TEST_FINISHED();
END_METHOD

METHOD PRIVATE Test_ANY_STRING_Differ_2
VAR
    a : STRING := 'This is a string';
    b : STRING := 'This is b string';
END_VAR
TEST('Test_ANY_STRING_Differ_2');

AssertEquals(Expected := a,
             Actual := b,
             Message := 'Values differ');

TEST_FINISHED();
END_METHOD

METHOD PRIVATE Test_ANY_STRING_Equals
VAR
    a : STRING := 'Hello there';
    b : STRING := 'Hello there';
END_VAR
TEST('Test_ANY_STRING_Equals');

AssertEquals(Expected := a,
             Actual := b,
             Message := 'Values differ');

TEST_FINISHED();
END_METHOD

METHOD PRIVATE Test_ANY_TIME_Differ
VAR
    a : TIME := T#12H34M15S10MS;
    b : TIME := T#11H34M13S244MS;
END_VAR
TEST('Test_ANY_TIME_Differ');

AssertEquals(Expected := a,
             Actual := b,
             Message := 'Values differ');

TEST_FINISHED();
END_METHOD

METHOD PRIVATE Test_ANY_TIME_Equals
VAR
    a : TIME := T#11H34M13S244MS;
    b : TIME := T#11H34M13S244MS;
END_VAR
TEST('Test_ANY_TIME_Equals');

AssertEquals(Expected := a,
             Actual := b,
             Message := 'Values differ');

TEST_FINISHED();
END_METHOD

METHOD PRIVATE Test_ANY_TIME_OF_DAY_Differ
VAR
    a : TIME_OF_DAY := TIME_OF_DAY#15:36:30.123;
    b : TIME_OF_DAY := TIME_OF_DAY#06:21:11.492;
END_VAR
TEST('Test_ANY_TIME_OF_DAY_Differ');

AssertEquals(Expected := a,
             Actual := b,
             Message := 'Values differ');

TEST_FINISHED();
END_METHOD

METHOD PRIVATE Test_ANY_TIME_OF_DAY_Equals
VAR
    a : TIME_OF_DAY := TIME_OF_DAY#06:21:11.492;
    b : TIME_OF_DAY := TIME_OF_DAY#06:21:11.492;
END_VAR
TEST('Test_ANY_TIME_OF_DAY_Equals');

AssertEquals(Expected := a,
             Actual := b,
             Message := 'Values differ');

TEST_FINISHED();
END_METHOD

METHOD PRIVATE Test_ANY_UDINT_Differ
VAR
    a : UDINT := 34124214;
    b : UDINT := 52343244;
END_VAR
TEST('Test_ANY_UDINT_Differ');

AssertEquals(Expected := a,
             Actual := b,
             Message := 'Values differ');

TEST_FINISHED();
END_METHOD

METHOD PRIVATE Test_ANY_UDINT_Equals
VAR
    a : UDINT := 21845123;
    b : UDINT := 21845123;
END_VAR
TEST('Test_ANY_UDINT_Equals');

AssertEquals(Expected := a,
             Actual := b,
             Message := 'Values differ');

TEST_FINISHED();
END_METHOD

METHOD PRIVATE Test_ANY_UINT_Differ
VAR
    a : UINT := 64322;
    b : UINT := 32312;
END_VAR
TEST('Test_ANY_UINT_Differ');

AssertEquals(Expected := a,
             Actual := b,
             Message := 'Values differ');

TEST_FINISHED();
END_METHOD

METHOD PRIVATE Test_ANY_UINT_Equals
VAR
    a : UINT := 65535;
    b : UINT := 65535;
END_VAR
TEST('Test_ANY_UINT_Equals');

AssertEquals(Expected := a,
             Actual := b,
             Message := 'Values differ');

TEST_FINISHED();
END_METHOD

METHOD PRIVATE Test_ANY_ULINT_Differ
VAR
    a : ULINT := 10000;
    b : ULINT := 53685437234;
END_VAR
TEST('Test_ANY_ULINT_Differ');

AssertEquals(Expected := a,
             Actual := b,
             Message := 'Values differ');

TEST_FINISHED();
END_METHOD

METHOD PRIVATE Test_ANY_ULINT_Equals
VAR
    a : ULINT := 45683838383;
    b : ULINT := 45683838383;
END_VAR
TEST('Test_ANY_ULINT_Equals');

AssertEquals(Expected := a,
             Actual := b,
             Message := 'Values differ');

TEST_FINISHED();
END_METHOD

METHOD PRIVATE Test_ANY_USINT_Differ
VAR
    a : USINT := 3;
    b : USINT := 7;
END_VAR
TEST('Test_ANY_USINT_Differ');

AssertEquals(Expected := a,
             Actual := b,
             Message := 'Values differ');

TEST_FINISHED();
END_METHOD

METHOD PRIVATE Test_ANY_USINT_Equals
VAR
    a : USINT := 5;
    b : USINT := 5;
END_VAR
TEST('Test_ANY_USINT_Equals');

AssertEquals(Expected := a,
             Actual := b,
             Message := 'Values differ');

TEST_FINISHED();
END_METHOD

METHOD PRIVATE Test_ANY_WORD_Differ
VAR
    a : WORD := 16#EF01;
    b : WORD := 16#2345;
END_VAR
TEST('Test_ANY_WORD_Differ');

AssertEquals(Expected := a,
             Actual := b,
             Message := 'Values differ');

TEST_FINISHED();
END_METHOD

METHOD PRIVATE Test_ANY_WORD_Equals
VAR
    a : WORD := 16#ABCD;
    b : WORD := 16#ABCD;
END_VAR
TEST('Test_ANY_WORD_Equals');

AssertEquals(Expected := a,
             Actual := b,
             Message := 'Values differ');

TEST_FINISHED();
END_METHOD

METHOD PRIVATE Test_ANY_WSTRING_Differ
VAR
    a : WSTRING := "äö";
    b : WSTRING := "æå";
END_VAR
TEST('Test_ANY_WSTRING_Differ');

AssertEquals(Expected := a,
             Actual := b,
             Message := 'Values differ');

TEST_FINISHED();
END_METHOD

METHOD PRIVATE Test_ANY_WSTRING_Differ_2
VAR
    a : WSTRING := "äö◦";
    b : WSTRING := "æå";
END_VAR
TEST('Test_ANY_WSTRING_Differ_2');

AssertEquals(Expected := a,
             Actual := b,
             Message := 'Values differ');

TEST_FINISHED();
END_METHOD

METHOD PRIVATE Test_ANY_WSTRING_Equals
VAR
    a : WSTRING := "ĠĦ";
    b : WSTRING := "ĠĦ";
END_VAR
TEST('Test_ANY_WSTRING_Equals');

AssertEquals(Expected := a,
             Actual := b,
             Message := 'Values differ');

TEST_FINISHED();
END_METHOD

END_FUNCTION_BLOCK

// ---- Test/FB_AssertEveryFailedTestTwiceArrayVersion.TcPOU
(*
    In this testsuite we are running the same testcase over two cycles, and thus calling
    every assert method twice. This is in order to verify that we don't print every FAILED assert twice.
    With this version we are doing it with arrays.
*)
FUNCTION_BLOCK FB_AssertEveryFailedTestTwiceArrayVersion EXTENDS TcUnit.FB_TestSuite
VAR
    AssertCount : USINT := 0;
END_VAR

TwiceAssertCall_Arrays();

METHOD PRIVATE TwiceAssertCall_Arrays
VAR
    aBOOL : ARRAY[0..5] OF BOOL := [TRUE, TRUE, FALSE, TRUE, FALSE, TRUE];
    bBOOL : ARRAY[0..5] OF BOOL := [TRUE, TRUE, TRUE, TRUE, FALSE, FALSE];

    aBYTE : ARRAY[0..3] OF BYTE := [16#AB, 16#AA, 16#BB, 16#89];
    bBYTE : ARRAY[0..3] OF BYTE := [16#AB, 16#CD, 16#BB, 16#89];

    aDINT : ARRAY[3..5] OF DINT := [-4746, -2147483645, 0];
    bDINT : ARRAY[3..5] OF DINT := [-4746, -2147483641, 0];

    aDWORD : ARRAY[-2..1] OF DWORD := [16#6789ABCD, 16#EFAA2346, 16#ABABABAB, 16#EEEEEEEE];
    bDWORD : ARRAY[-2..1] OF DWORD := [16#6789ABCD, 16#EF012345, 16#ABABABAB, 16#EEEEEEEE];

    aINT : ARRAY[-8..-6] OF INT := [42, -23, -32768];
    bINT : ARRAY[1..3] OF INT := [42, 24, -32768];

    aLINT : ARRAY[-1..1] OF LINT := [9_223_372_036_854_775_807, -9_223_372_036_853_775_808, 55];
    bLINT : ARRAY[4..6] OF LINT := [9_223_372_036_854_775_807, -9_223_372_036_854_775_808, 55];

    aLREAL : ARRAY[-2..1] OF LREAL := [3.55, 7.88, 2.44];
    bLREAL : ARRAY[-1..2] OF LREAL := [3.56, 7.99, 2.44];

    aLREAL2d : ARRAY[0..1, 0..1] OF LREAL := [4.44, 5.75, 6.96, 7.77];
    bLREAL2d : ARRAY[0..1, 0..1] OF LREAL := [4.45, 5.75, 6.68, 7.77];

    aLREAL3d : ARRAY[0..1, 0..1, 0..1] OF LREAL := [1.0, 2.0, 3.0, 4.0, 5.0, 6.0, 7.0, 8.0];
    bLREAL3d : ARRAY[0..1, 0..1, 0..1] OF LREAL := [1.0, 2.0, 3.0, 4.0, 5.0, 6.4, 7.0, 8.0];

    aLWORD : ARRAY[1..1] OF LWORD := [16#EDCBA09876543210];
    bLWORD : ARRAY[1..1] OF LWORD := [16#01234567890ABCDE];

    aREAL : ARRAY[0..2] OF REAL := [6.55000001, 3.54, 2.44001];
    bREAL : ARRAY[0..2] OF REAL := [6.55, 3.54, 2.44003];

    aREAL2d : ARRAY[0..1, 0..1] OF REAL := [4.45, 5.75, 6.960001, 7.7701];
    bREAL2d : ARRAY[0..1, 0..1] OF REAL := [4.45, 5.75, 6.960002, 7.7703];

    aREAL3d : ARRAY[0..1, 0..1, 0..1] OF REAL := [1.0, 2.0, 3.0, 4.01, 5.0, 6.0, 7.0, 8.0];
    bREAL3d : ARRAY[0..1, 0..1, 0..1] OF REAL := [1.0, 2.0, 3.0, 4.021, 5.0, 6.0, 7.0, 8.0];

    aSINT : ARRAY[0..0] OF SINT := [-128];
    bSINT : ARRAY[0..0] OF SINT := [127];

    aUDINT : ARRAY[-5..-4] OF UDINT := [4294967295, 5];
    bUDINT : ARRAY[0..1] OF UDINT := [4294967295, 4];

    aUINT : ARRAY[0..3] OF UINT := [0, 4, 8, 99];
    bUINT : ARRAY[0..3] OF UINT := [0, 4, 8, 12];

    aULINT : ARRAY[0..1] OF ULINT := [3_213_000_444_000, 9_400_000_000_000];
    bULINT : ARRAY[0..1] OF ULINT := [3_213_000_444_000, 18_446_744_073_709_551_615];

    aUSINT : ARRAY[0..10] OF USINT := [0,1,2,3,6(4),5];
    bUSINT : ARRAY[0..10] OF USINT := [0,1,2,3,6(5),6];

    aWORD : ARRAY[1..7] OF WORD := [16#2323, 16#876A, 16#4CD4, 16#F3DC, 16#BBBB, 16#FFFF, 16#1133];
    bWORD : ARRAY[1..7] OF WORD := [16#2323, 16#876A, 16#4CD4, 16#F3DC, 16#BBBB, 16#FFFF, 16#1122];
END_VAR
TEST('TwiceAssertCall_Arrays');

AssertArrayEquals_BOOL(Expecteds := aBOOL,
                       Actuals := bBOOL,
                       Message := 'Not equal BOOL');

AssertArrayEquals_BYTE(Expecteds := aBYTE,
                       Actuals := bBYTE,
                       Message := 'Not equal BYTE');

AssertArrayEquals_DINT(Expecteds := aDINT,
                       Actuals := bDINT,
                       Message := 'Not equal DINT');

AssertArrayEquals_DWORD(Expecteds := aDWORD,
                        Actuals := bDWORD,
                        Message := 'Not equal DWORD');

AssertArrayEquals_INT(Expecteds := aINT,
                      Actuals := bINT,
                      Message := 'Not equal INT');

AssertArrayEquals_LINT(Expecteds := aLINT,
                       Actuals := bLINT,
                       Message := 'Not equal LINT');

AssertArrayEquals_LREAL(Expecteds := aLREAL,
                        Actuals := bLREAL,
                        Delta := 0.1,
                        Message := 'Not equal LREAL');

AssertArray2dEquals_LREAL(Expecteds := aLREAL2d,
                          Actuals := bLREAL2d,
                          Delta := 0.1,
                          Message := 'Not equal LREAL2D');

AssertArray3dEquals_LREAL(Expecteds := aLREAL3d,
                          Actuals := bLREAL3d,
                          Delta := 0.1,
                          Message := 'Not equal LREAL3D');

AssertArrayEquals_LWORD(Expecteds := aLWORD,
                        Actuals := bLWORD,
                        Message := 'Not equal LWORD');

AssertArrayEquals_SINT(Expecteds := aSINT,
                       Actuals := bSINT,
                       Message := 'Not equal SINT');

AssertArrayEquals_REAL(Expecteds := aREAL,
                       Actuals := bREAL,
                       Delta := 0.00001,
                       Message := 'Not equal REAL');

AssertArray2dEquals_REAL(Expecteds := aREAL2d,
                         Actuals := bREAL2d,
                         Delta := 0.0001,
                         Message := 'Not equal REAL2D');

AssertArray3dEquals_REAL(Expecteds := aREAL3d,
                         Actuals := bREAL3d,
                         Delta := 0.01,
                         Message := 'Not equal REAL3D');

AssertArrayEquals_UDINT(Expecteds := aUDINT,
                        Actuals := bUDINT,
                        Message := 'Not equal UDINT');

AssertArrayEquals_UINT(Expecteds := aUINT,
                       Actuals := bUINT,
                       Message := 'Not equal UINT');

AssertArrayEquals_ULINT(Expecteds := aULINT,
                        Actuals := bULINT,
                        Message := 'Not equal ULINT');

AssertArrayEquals_USINT(Expecteds := aUSINT,
                        Actuals := bUSINT,
                        Message := 'Not equal USINT');

AssertArrayEquals_WORD(Expecteds := aWORD,
                       Actuals := bWORD,
                       Message := 'Not equal WORD');

AssertCount := AssertCount + 1;
IF AssertCount = 2 THEN
    TEST_FINISHED();
END_IF
END_METHOD

END_FUNCTION_BLOCK

// ---- Test/FB_AnyToUnionValue.TcPOU
(*
    Tests the free function F_AnyToUnionValue.
*)
FUNCTION_BLOCK FB_AnyToUnionValue EXTENDS TcUnit.FB_TestSuite
VAR
    aBit : BIT := 1; // Only structures and function blocks can have BIT defined
END_VAR

Test_BOOL();
Test_BIT();
Test_BYTE();
Test_WORD();
Test_DWORD();
Test_LWORD();
Test_SINT();
Test_INT();
Test_DINT();
Test_LINT();
Test_USINT();
Test_UINT();
Test_UDINT();
Test_ULINT();
Test_REAL();
Test_LREAL();
Test_STRING();
Test_STRING_2();
Test_WSTRING();
Test_TIME();
Test_DATE();
Test_DATE_AND_TIME();
Test_TIME_OF_DAY();
Test_LTIME();

METHOD PRIVATE Test_BIT
VAR
    Result : U_ExpectedOrActual;
END_VAR
TEST('Test_BIT');

Result := TcUnit.F_AnyToUnionValue(AnySize := SIZEOF(aBit), AnyTypeClass := IBaseLibrary.TYPE_BIT, AnyValue := ADR(aBit));

AssertEquals(Expected := aBit,
             Actual := result.bitExpectedOrActual,
             Message := 'Values differ');

TEST_FINISHED();
END_METHOD

METHOD PRIVATE Test_BOOL
VAR
    a : BOOL := TRUE;
    Result : U_ExpectedOrActual;
END_VAR
TEST('Test_BOOL');

Result := TcUnit.F_AnyToUnionValue(AnySize := SIZEOF(a), AnyTypeClass := IBaseLibrary.TYPE_BOOL, AnyValue := ADR(a));

AssertEquals(Expected := a,
             Actual := result.boolExpectedOrActual,
             Message := 'Values differ');

TEST_FINISHED();
END_METHOD

METHOD PRIVATE Test_BYTE
VAR
    a : BYTE := 16#8A;
    Result : U_ExpectedOrActual;
END_VAR
TEST('Test_BYTE');

Result := TcUnit.F_AnyToUnionValue(AnySize := SIZEOF(a), AnyTypeClass := IBaseLibrary.TYPE_BYTE, AnyValue := ADR(a));

AssertEquals(Expected := a,
             Actual := result.byteExpectedOrActual,
             Message := 'Values differ');

TEST_FINISHED();
END_METHOD

METHOD PRIVATE Test_DATE
VAR
    a : DATE := D#2106-02-05;
    Result : U_ExpectedOrActual;
END_VAR
TEST('Test_DATE');

Result := TcUnit.F_AnyToUnionValue(AnySize := SIZEOF(a), AnyTypeClass := IBaseLibrary.TYPE_DATE, AnyValue := ADR(a));

AssertEquals(Expected := a,
             Actual := result.dateExpectedOrActual,
             Message := 'Values differ');

TEST_FINISHED();
END_METHOD

METHOD PRIVATE Test_DATE_AND_TIME
VAR
    a : DATE_AND_TIME := DT#2106-02-06-06:28:15;
    Result : U_ExpectedOrActual;
END_VAR
TEST('Test_DATE_AND_TIME');

Result := TcUnit.F_AnyToUnionValue(AnySize := SIZEOF(a), AnyTypeClass := IBaseLibrary.TYPE_DATEANDTIME, AnyValue := ADR(a));

AssertEquals(Expected := a,
             Actual := result.dateandtimeExpectedOrActual,
             Message := 'Values differ');

TEST_FINISHED();
END_METHOD

METHOD PRIVATE Test_DINT
VAR
    a : DINT := 143251;
    Result : U_ExpectedOrActual;
END_VAR
TEST('Test_DINT');

Result := TcUnit.F_AnyToUnionValue(AnySize := SIZEOF(a), AnyTypeClass := IBaseLibrary.TYPE_DINT, AnyValue := ADR(a));

AssertEquals(Expected := a,
             Actual := result.dintExpectedOrActual,
             Message := 'Values differ');

TEST_FINISHED();
END_METHOD

METHOD PRIVATE Test_DWORD
VAR
    a : DWORD := 16#3456CDEF;
    Result : U_ExpectedOrActual;
END_VAR
TEST('Test_DWORD');

Result := TcUnit.F_AnyToUnionValue(AnySize := SIZEOF(a), AnyTypeClass := IBaseLibrary.TYPE_DWORD, AnyValue := ADR(a));

AssertEquals(Expected := a,
             Actual := result.dwordExpectedOrActual,
             Message := 'Values differ');

TEST_FINISHED();
END_METHOD

METHOD PRIVATE Test_INT
VAR
    a : INT := -32000;
    Result : U_ExpectedOrActual;
END_VAR
TEST('Test_INT');

Result := TcUnit.F_AnyToUnionValue(AnySize := SIZEOF(a), AnyTypeClass := IBaseLibrary.TYPE_INT, AnyValue := ADR(a));

AssertEquals(Expected := a,
             Actual := result.intExpectedOrActual,
             Message := 'Values differ');

TEST_FINISHED();
END_METHOD

METHOD PRIVATE Test_LINT
VAR
    a : LINT := -31243145;
    Result : U_ExpectedOrActual;
END_VAR
TEST('Test_LINT');

Result := TcUnit.F_AnyToUnionValue(AnySize := SIZEOF(a), AnyTypeClass := IBaseLibrary.TYPE_LINT, AnyValue := ADR(a));

AssertEquals(Expected := a,
             Actual := result.lintExpectedOrActual,
             Message := 'Values differ');

TEST_FINISHED();
END_METHOD

METHOD PRIVATE Test_LREAL
VAR
    a : LREAL := 43123923124.745423;
    Result : U_ExpectedOrActual;
END_VAR
TEST('Test_LREAL');

Result := TcUnit.F_AnyToUnionValue(AnySize := SIZEOF(a), AnyTypeClass := IBaseLibrary.TYPE_LREAL, AnyValue := ADR(a));

AssertEquals(Expected := a,
             Actual := result.lrealExpectedOrActual,
             Message := 'Values differ');

TEST_FINISHED();
END_METHOD

METHOD PRIVATE Test_LTIME
VAR
    a : LTIME := LTIME#213502D23H34M33S709MS551US615NS;
    Result : U_ExpectedOrActual;
END_VAR
TEST('Test_LTIME');

Result := TcUnit.F_AnyToUnionValue(AnySize := SIZEOF(a), AnyTypeClass := IBaseLibrary.TYPE_LTIME, AnyValue := ADR(a));

AssertEquals(Expected := a,
             Actual := result.ltimeExpectedOrActual,
             Message := 'Values differ');

TEST_FINISHED();
END_METHOD

METHOD PRIVATE Test_LWORD
VAR
    a : LWORD := 16#456CDEF987654321;
    Result : U_ExpectedOrActual;
END_VAR
TEST('Test_LWORD');

Result := TcUnit.F_AnyToUnionValue(AnySize := SIZEOF(a), AnyTypeClass := IBaseLibrary.TYPE_LWORD, AnyValue := ADR(a));

AssertEquals(Expected := a,
             Actual := result.lwordExpectedOrActual,
             Message := 'Values differ');

TEST_FINISHED();
END_METHOD

METHOD PRIVATE Test_REAL
VAR
    a : REAL := 431239.423;
    Result : U_ExpectedOrActual;
END_VAR
TEST('Test_REAL');

Result := TcUnit.F_AnyToUnionValue(AnySize := SIZEOF(a), AnyTypeClass := IBaseLibrary.TYPE_REAL, AnyValue := ADR(a));

AssertEquals(Expected := a,
             Actual := result.realExpectedOrActual,
             Message := 'Values differ');

TEST_FINISHED();
END_METHOD

METHOD PRIVATE Test_SINT
VAR
    a : SINT := 100;
    Result : U_ExpectedOrActual;
END_VAR
TEST('Test_SINT');

Result := TcUnit.F_AnyToUnionValue(AnySize := SIZEOF(a), AnyTypeClass := IBaseLibrary.TYPE_SINT, AnyValue := ADR(a));

AssertEquals(Expected := a,
             Actual := result.sintExpectedOrActual,
             Message := 'Values differ');

TEST_FINISHED();
END_METHOD

METHOD PRIVATE Test_STRING
VAR
    a : STRING := 'This is a random string';
    Result : U_ExpectedOrActual;
END_VAR
TEST('Test_STRING');

Result := TcUnit.F_AnyToUnionValue(AnySize := SIZEOF(a), AnyTypeClass := IBaseLibrary.TYPE_STRING, AnyValue := ADR(a));

AssertEquals(Expected := a,
             Actual := result.stringExpectedOrActual,
             Message := 'Values differ');

TEST_FINISHED();
END_METHOD

METHOD PRIVATE Test_STRING_2
VAR
    a : T_MaxString := '8YNn5KOmPC4dAcpOBdLWnw4WkN126EwXsj65xeurG48gWBepinNaOIKeCVMtWNBSxQWPdtUYiAusDkjMLtQhDtiWbwvmoKcFwiUGDd7pOe0fd52J7hK60oaYAX6VWWmceLJX8utaDVrVzCGXafeZLeHl6jj5enfjg4tfb2WMEBdsBuG2iDKwzwhBLCPqXDnhe5HbemIbtZT7p62OEj2oDqiIYDD6tZdlhBCCelDBx6dbIp32wFm0TpRKsTiwkZ6'; // 255 characters
    Result : U_ExpectedOrActual;
END_VAR
TEST('Test_STRING_2');

Result := TcUnit.F_AnyToUnionValue(AnySize := SIZEOF(a), AnyTypeClass := IBaseLibrary.TYPE_STRING, AnyValue := ADR(a));

AssertEquals(Expected := a,
             Actual := result.stringExpectedOrActual,
             Message := 'Values differ');

TEST_FINISHED();
END_METHOD

METHOD PRIVATE Test_TIME
VAR
    a : TIME := T#15M20S;
    Result : U_ExpectedOrActual;
END_VAR
TEST('Test_TIME');

Result := TcUnit.F_AnyToUnionValue(AnySize := SIZEOF(a), AnyTypeClass := IBaseLibrary.TYPE_TIME, AnyValue := ADR(a));

AssertEquals(Expected := a,
             Actual := result.timeExpectedOrActual,
             Message := 'Values differ');

TEST_FINISHED();
END_METHOD

METHOD PRIVATE Test_TIME_OF_DAY
VAR
    a : TIME_OF_DAY := TOD#15:36:30.123;
    Result : U_ExpectedOrActual;
END_VAR
TEST('Test_TIME_OF_DAY');

Result := TcUnit.F_AnyToUnionValue(AnySize := SIZEOF(a), AnyTypeClass := IBaseLibrary.TYPE_TIMEOFDAY, AnyValue := ADR(a));

AssertEquals(Expected := a,
             Actual := result.timeofdayExpectedOrActual,
             Message := 'Values differ');

TEST_FINISHED();
END_METHOD

METHOD PRIVATE Test_UDINT
VAR
    a : UDINT := 2555;
    Result : U_ExpectedOrActual;
END_VAR
TEST('Test_UDINT');

Result := TcUnit.F_AnyToUnionValue(AnySize := SIZEOF(a), AnyTypeClass := IBaseLibrary.TYPE_UDINT, AnyValue := ADR(a));

AssertEquals(Expected := a,
             Actual := result.udintExpectedOrActual,
             Message := 'Values differ');

TEST_FINISHED();
END_METHOD

METHOD PRIVATE Test_UINT
VAR
    a : UINT := 34523;
    Result : U_ExpectedOrActual;
END_VAR
TEST('Test_UINT');

Result := TcUnit.F_AnyToUnionValue(AnySize := SIZEOF(a), AnyTypeClass := IBaseLibrary.TYPE_UINT, AnyValue := ADR(a));

AssertEquals(Expected := a,
             Actual := result.uintExpectedOrActual,
             Message := 'Values differ');

TEST_FINISHED();
END_METHOD

METHOD PRIVATE Test_ULINT
VAR
    a : ULINT := 25555423;
    Result : U_ExpectedOrActual;
END_VAR
TEST('TEST_ULINT');

Result := TcUnit.F_AnyToUnionValue(AnySize := SIZEOF(a), AnyTypeClass := IBaseLibrary.TYPE_ULINT, AnyValue := ADR(a));

AssertEquals(Expected := a,
             Actual := result.ulintExpectedOrActual,
             Message := 'Values differ');

TEST_FINISHED();
END_METHOD

METHOD PRIVATE Test_USINT
VAR
    a : USINT := 255;
    Result : U_ExpectedOrActual;
END_VAR
TEST('Test_USINT');

Result := TcUnit.F_AnyToUnionValue(AnySize := SIZEOF(a), AnyTypeClass := IBaseLibrary.TYPE_USINT, AnyValue := ADR(a));

AssertEquals(Expected := a,
             Actual := result.usintExpectedOrActual,
             Message := 'Values differ');

TEST_FINISHED();
END_METHOD

METHOD PRIVATE Test_WORD
VAR
    a : WORD := 16#ABCD;
    Result : U_ExpectedOrActual;
END_VAR
TEST('Test_WORD');

Result := TcUnit.F_AnyToUnionValue(AnySize := SIZEOF(a), AnyTypeClass := IBaseLibrary.TYPE_WORD, AnyValue := ADR(a));

AssertEquals(Expected := a,
             Actual := result.wordExpectedOrActual,
             Message := 'Values differ');

TEST_FINISHED();
END_METHOD

METHOD PRIVATE Test_WSTRING
VAR
    a : WSTRING := "åäöĦ";
    Result : U_ExpectedOrActual;
END_VAR
TEST('Test_WSTRING');

Result := TcUnit.F_AnyToUnionValue(AnySize := SIZEOF(a), AnyTypeClass := IBaseLibrary.TYPE_WSTRING, AnyValue := ADR(a));

AssertEquals(Expected := a,
             Actual := result.wstringExpectedOrActual,
             Message := 'Values differ');

TEST_FINISHED();
END_METHOD

END_FUNCTION_BLOCK

// ---- Test/FB_MultipleAssertWithSameParametersInSameCycleWithSameTest.TcPOU
(*
    This test-suite runs several asserts with the same parameters (same expected, actual, message) in the same cycle
    and in the same test.
    The reason we want the framework to support this is that theoretically the user could want to do an assert with the
    same message, in the same test, with the same data values for both expected and actual, although the data that the
    user does the assert on might be from different data sets.
*)
FUNCTION_BLOCK FB_MultipleAssertWithSameParametersInSameCycleWithSameTest EXTENDS TcUnit.FB_TestSuite

Assert_SeveralTimes();

METHOD PRIVATE Assert_SeveralTimes
VAR
    a : DWORD := 16#12345678;
    b : DWORD := 16#90ABCDEF;

    c : DWORD := 16#12345678;
    d : DWORD := 16#90ABCDEF;

    e : DWORD := 16#12345678;
    f : DWORD := 16#90ABCDEF;
END_VAR
TEST('Assert_SeveralTimes');

AssertEquals_DWORD(Expected := a,
                   Actual := b,
                   Message := 'Values differ');

AssertEquals_DWORD(Expected := c,
                   Actual := d,
                   Message := 'Values differ');

AssertEquals_DWORD(Expected := e,
                   Actual := f,
                   Message := 'Values differ');

TEST_FINISHED();
END_METHOD

END_FUNCTION_BLOCK

// ---- Test/FB_MultipleAssertWithSameParametersInDifferentCyclesButWithDifferentTests.TcPOU
(*
    This test-suite runs several asserts with the same parameters (same expected, actual, message), calling the asserts
    in different cycles and using different tests.
    On top of this, we will call new asserts (though with same parameters) in later cycles.
    The reason we want the framework to support this is that theoretically the user could want to do an assert with the
    same message, in different tests, with the same data values for both expected and actual, although the data that the
    user does the assert on might be from different data sets.
*)
FUNCTION_BLOCK FB_MultipleAssertWithSameParametersInDifferentCyclesButWithDifferentTests EXTENDS TcUnit.FB_TestSuite
VAR
    TimerAgain : TON := (PT := T#1S); // Timer to call "AssertSeveralTimesAgain"
    TimerAgainAgain : TON := (PT := T#5S); // Timer to call "AssertSeveralTimesAgainAgain"
    CalledAll : BOOL; // Indication of whether we've called all tests
END_VAR

TimerAgain(IN := TRUE);

Assert_SeveralTimes();

IF TimerAgain.Q THEN
    TimerAgainAgain(IN := TRUE);
    Assert_SeveralTimesAgain();
END_IF

IF TimerAgainAgain.Q THEN
    Assert_SeveralTimesAgainAgain();
    CalledAll := TRUE;
END_IF

METHOD PRIVATE Assert_SeveralTimes
VAR
    a : DWORD := 16#12345678;
    b : DWORD := 16#90ABCDEF;

    c : DWORD := 16#12345678;
    d : DWORD := 16#90ABCDEF;

    e : DWORD := 16#12345678;
    f : DWORD := 16#90ABCDEF;
END_VAR
TEST('Assert_SeveralTimes');

AssertEquals_DWORD(Expected := a,
                   Actual := b,
                   Message := 'Values differ');

AssertEquals_DWORD(Expected := c,
                   Actual := d,
                   Message := 'Values differ');

AssertEquals_DWORD(Expected := e,
                   Actual := f,
                   Message := 'Values differ');

IF CalledAll THEN
    TEST_FINISHED();
END_IF
END_METHOD

METHOD PRIVATE Assert_SeveralTimesAgain
VAR
    a : DWORD := 16#12345678;
    b : DWORD := 16#90ABCDEF;

    c : DWORD := 16#12345678;
    d : DWORD := 16#90ABCDEF;

    e : DWORD := 16#12345678;
    f : DWORD := 16#90ABCDEF;
END_VAR
TEST('Assert_SeveralTimesAgain');

AssertEquals_DWORD(Expected := a,
                   Actual := b,
                   Message := 'Values differ');

AssertEquals_DWORD(Expected := c,
                   Actual := d,
                   Message := 'Values differ');

AssertEquals_DWORD(Expected := e,
                   Actual := f,
                   Message := 'Values differ');

IF CalledAll THEN
    TEST_FINISHED();
END_IF
END_METHOD

METHOD PRIVATE Assert_SeveralTimesAgainAgain
VAR
    a : DWORD := 16#12345678;
    b : DWORD := 16#90ABCDEF;

    c : DWORD := 16#12345678;
    d : DWORD := 16#90ABCDEF;

    e : DWORD := 16#12345678;
    f : DWORD := 16#90ABCDEF;
END_VAR
TEST('Assert_SeveralTimesAgainAgain');

AssertEquals_DWORD(Expected := a,
                   Actual := b,
                   Message := 'Values differ');

AssertEquals_DWORD(Expected := c,
                   Actual := d,
                   Message := 'Values differ');

AssertEquals_DWORD(Expected := e,
                   Actual := f,
                   Message := 'Values differ');

IF CalledAll THEN
    TEST_FINISHED();
END_IF
END_METHOD

END_FUNCTION_BLOCK

// ---- Test/FB_MultipleAssertWithSameParametersInDifferentCyclesAndInSameTest.TcPOU
(*
    This test-suite runs several asserts with the same parameters (same expected, actual, message), calling the asserts
    in different cycles and using the same test.
    On top of this, we will call new asserts (though with same parameters) in later cycles.
    The reason we want the framework to support this is that theoretically the user could want to do an assert with the
    same message, using the same test with the same data values for both expected and actual, and splitting the asserts
    on different cycles.
*)
FUNCTION_BLOCK FB_MultipleAssertWithSameParametersInDifferentCyclesAndInSameTest EXTENDS TcUnit.FB_TestSuite
VAR
    TimerAgain : TON := (PT := T#1S); // Timer to call "AssertSeveralTimesAgain"
    TimerAgainAgain : TON := (PT := T#5S); // Timer to call "AssertSeveralTimesAgainAgain"
    CalledAll : BOOL; // Indication of whether we've called all tests
END_VAR

Assert_SeveralTimes();

METHOD PRIVATE Assert_SeveralTimes
VAR
    a : DWORD := 16#12345678;
    b : DWORD := 16#90ABCDEF;

    c : DWORD := 16#12345678;
    d : DWORD := 16#90ABCDEF;

    e : DWORD := 16#12345678;
    f : DWORD := 16#90ABCDEF;

    g : DWORD := 16#12345678;
    h : DWORD := 16#90ABCDEF;

    i : DWORD := 16#12345678;
    j : DWORD := 16#90ABCDEF;

    k : DWORD := 16#12345678;
    l : DWORD := 16#90ABCDEF;

    m : DWORD := 16#12345678;
    n : DWORD := 16#90ABCDEF;

    o : DWORD := 16#12345678;
    p : DWORD := 16#90ABCDEF;

    q : DWORD := 16#12345678;
    rr : DWORD := 16#90ABCDEF;
END_VAR
TEST('Assert_SeveralTimes');

AssertEquals_DWORD(Expected := a,
                   Actual := b,
                   Message := 'Values differ');
AssertEquals_DWORD(Expected := c,
                   Actual := d,
                   Message := 'Values differ');
AssertEquals_DWORD(Expected := e,
                   Actual := f,
                   Message := 'Values differ');

TimerAgain(IN := TRUE);
IF TimerAgain.Q THEN
    TimerAgainAgain(IN := TRUE);
    AssertEquals_DWORD(Expected := g,
                       Actual := h,
                       Message := 'Values differ');
    AssertEquals_DWORD(Expected := i,
                       Actual := j,
                       Message := 'Values differ');
    AssertEquals_DWORD(Expected := k,
                       Actual := l,
                       Message := 'Values differ');
END_IF

IF TimerAgainAgain.Q THEN
    AssertEquals_DWORD(Expected := m,
                       Actual := n,
                       Message := 'Values differ');
    AssertEquals_DWORD(Expected := o,
                       Actual := p,
                       Message := 'Values differ');
    AssertEquals_DWORD(Expected := q,
                       Actual := rr,
                       Message := 'Values differ');
    CalledAll := TRUE;
    TEST_FINISHED();
END_IF
END_METHOD

END_FUNCTION_BLOCK

// ---- Test/FB_SkipAssertionsWhenFinished.TcPOU
(*
    Contains tests that require multiple cycles:
    - A short test that finishes quickly
        - The assert statements all pass while the test is not finished
        - After the test is finished, the variables change so that the assert statements now fail,
            which shouldn't matter because the test is finished
    - A long test that finishes slowly
        - This test exists so that the entire test suite keeps running after the short test finishes
*)
FUNCTION_BLOCK FB_SkipAssertionsWhenFinished EXTENDS TcUnit.FB_TestSuite
VAR
    ShortTimer : TON := (PT := T#200MS);
    LongTimer : TON := (PT := T#1S);
END_VAR

Test_LongTest(ADR(LongTimer));
Test_ShortTest(ADR(ShortTimer));
Test_AssertImmediatelyAfterFinished();

(*
    Assertions called immediately after (and within the same cycle as) TEST_FINISHED should be
    ignored.
*)
METHOD Test_AssertImmediatelyAfterFinished
TEST('Test_AssertImmediatelyAfterFinished');
TEST_FINISHED();

AssertTrue(FALSE, 'This failing assertion should be skipped because the test is finished');
END_METHOD

METHOD Test_LongTest
VAR_INPUT
    Timer : POINTER TO TON;
END_VAR
TEST('Test_LongTest');

Timer^(IN := TRUE);
IF Timer^.Q THEN
    TEST_FINISHED();
END_IF
END_METHOD

METHOD Test_ShortTest
VAR_INPUT
    Timer : POINTER TO TON;
END_VAR
TEST('Test_ShortTest');

AssertFalse(Timer^.Q, 'This assertion will start to fail after the test is over, but it will be skipped at that point');

Timer^(IN := TRUE);
IF Timer^.Q THEN
    TEST_FINISHED();
END_IF
END_METHOD

END_FUNCTION_BLOCK

// ---- Test/FB_AdjustAssertFailureMessageToMaxAllowedLengthTest.TcPOU
(* This testsuite tests the function block FB_AdjustAssertFailureMessageToMaxAllowedLength
   The total printed message can not be more than 250 characters long.
*)
FUNCTION_BLOCK FB_AdjustAssertFailureMessageToMaxAllowedLengthTest EXTENDS TcUnit.FB_TestSuite

TestInstancePath221CharsExpectShortenedTestInstancePath();
TestInstancePath252CharsExpectTooLongTestInstancePath();
TestInstancePath253CharsExpectTooLongTestInstancePath();
TestInstancePath255CharsExpectTooLongTestInstancePath();

METHOD TestInstancePath221CharsExpectShortenedTestInstancePath
VAR
    AdjustAssertFailureMessageToMaxAllowedLength : FB_AdjustAssertFailureMessageToMaxAllowedLength;

    // @Text-Fixture
    TestInstancePathNameWith221Chars : T_MaxString := 'PRG_TEST.LongInstanceNameLongInstanceNameLongInstanceNameLongInstanceNameLongInstanceNameLongInstanceNameLongInstanceNameLongInstanceNameLongInstanceNameLongInstanceName@LONGTESTNAMELONGTESTNAMELONGTESTNAMELONGTESTNAMELON';
    TooLongTestMessage60Chars : T_MaxString := 'Very long message that is 60 characters long which means tha';

    // @Test-Result-Expected
    // 220 + 32 = 252 (in other words, expected test message should be 32 characters long including '...TestMsg too long'
    TestMessageResultExpected : T_MaxString := 'Very long me...TestMsg too long'; 

    // @Test-Result
    TestInstancePathResult : T_MaxString;
    TestMessageResult : T_MaxString;
END_VAR
TEST('TestInstancePath221CharsExpectShortenedTestInstancePath');

AdjustAssertFailureMessageToMaxAllowedLength(TestInstancePath := TestInstancePathNameWith221Chars,
                                             TestMessage := TooLongTestMessage60Chars,
                                             TestInstancePathProcessed => TestInstancePathResult,
                                             TestMessageProcessed => TestMessageResult);

AssertEquals_STRING(Expected := TestInstancePathNameWith221Chars, // Same test instance path should be expected as the one going in
                    Actual := TestInstancePathResult,
                    'Test instance path not correct');

AssertEquals_STRING(Expected := TestMessageResultExpected,
                    Actual := TestMessageResult,
                    'Test message not correct');

TEST_FINISHED();
END_METHOD

METHOD PRIVATE TestInstancePath252CharsExpectTooLongTestInstancePath
VAR
    AdjustAssertFailureMessageToMaxAllowedLength : FB_AdjustAssertFailureMessageToMaxAllowedLength;

    // @Text-Fixture
    TestInstancePathNameWith252Chars : T_MaxString := 'PRG_TEST.LongInstanceNameLongInstanceNameLongInstanceNameLongInstanceNameLongInstanceNameLongInstanceNameLongInstanceNameLongInstanceNameLongInstanceNameLongInstanceName@LONGTESTNAMELONGTESTNAMELONGTESTNAMELONGTESTNAMELONGTESTNAMELONGTESTNAMELONGTESTNA';
    ShortTestMessage : T_MaxString := 'Very short message';

    // @Test-Result-Expected
    TestInstancePathNameWith252CharsExpectedResult : T_MaxString := 'PRG_TEST.LongInstanceNameLongInstanceNameLongInstanceNameLongInstanceNameLongInstanceNameLongInstanceNameLongInstanceNameLongInstanceNameLongInstanceNameLongInstanceName@LONGTESTNAMELONGTESTNAMELONGTESTNAMELONGTESTNAMELONGTESTNAMELO...TestName too long';
    ShortTestMessageExpectedResult : T_MaxString := '';

    // @Test-Result
    TestInstancePathNameWith252CharsResult : T_MaxString;
    ShortTestMessageResult : T_MaxString;
END_VAR
TEST('TestInstancePath252CharsExpectTooLongTestInstancePath');

AdjustAssertFailureMessageToMaxAllowedLength(TestInstancePath := TestInstancePathNameWith252Chars,
                                             TestMessage := ShortTestMessage,
                                             TestInstancePathProcessed => TestInstancePathNameWith252CharsResult,
                                             TestMessageProcessed => ShortTestMessageResult);

AssertEquals_STRING(Expected := TestInstancePathNameWith252CharsExpectedResult,
                    Actual := TestInstancePathNameWith252CharsResult,
                    'Test instance path not correct');

AssertEquals_STRING(Expected := ShortTestMessageExpectedResult,
                    Actual := ShortTestMessageResult,
                    'Test message not correct');

TEST_FINISHED();
END_METHOD

METHOD PRIVATE TestInstancePath253CharsExpectTooLongTestInstancePath
VAR
    AdjustAssertFailureMessageToMaxAllowedLength : FB_AdjustAssertFailureMessageToMaxAllowedLength;

    // @Text-Fixture
    TestInstancePathNameWith253Chars : T_MaxString := 'PRG_TEST.LongInstanceNameLongInstanceNameLongInstanceNameLongInstanceNameLongInstanceNameLongInstanceNameLongInstanceNameLongInstanceNameLongInstanceNameLongInstanceName@LONGTESTNAMELONGTESTNAMELONGTESTNAMELONGTESTNAMELONGTESTNAMELONGTESTNAMELONGTESTNAM';
    ShortTestMessage : T_MaxString := 'Very short message';

    // @Test-Result-Expected
    TestInstancePathNameWith252CharsExpectedResult : T_MaxString := 'PRG_TEST.LongInstanceNameLongInstanceNameLongInstanceNameLongInstanceNameLongInstanceNameLongInstanceNameLongInstanceNameLongInstanceNameLongInstanceNameLongInstanceName@LONGTESTNAMELONGTESTNAMELONGTESTNAMELONGTESTNAMELONGTESTNAMELO...TestName too long';
    ShortTestMessageExpectedResult : T_MaxString := '';

    // @Test-Result
    TestInstancePathNameWith252CharsResult : T_MaxString;
    ShortTestMessageResult : T_MaxString;
END_VAR
TEST('TestInstancePath253CharsExpectTooLongTestInstancePath');

AdjustAssertFailureMessageToMaxAllowedLength(TestInstancePath := TestInstancePathNameWith253Chars,
                                             TestMessage := ShortTestMessage,
                                             TestInstancePathProcessed => TestInstancePathNameWith252CharsResult,
                                             TestMessageProcessed => ShortTestMessageResult);

AssertEquals_STRING(Expected := TestInstancePathNameWith252CharsExpectedResult,
                    Actual := TestInstancePathNameWith252CharsResult,
                    'Test instance path not correct');

AssertEquals_STRING(Expected := ShortTestMessageExpectedResult,
                    Actual := ShortTestMessageResult,
                    'Test message not correct');

TEST_FINISHED();
END_METHOD

METHOD PRIVATE TestInstancePath255CharsExpectTooLongTestInstancePath
VAR
    AdjustAssertFailureMessageToMaxAllowedLength : FB_AdjustAssertFailureMessageToMaxAllowedLength;

    // @Text-Fixture
    TestInstancePathNameWith255Chars : T_MaxString := 'PRG_TEST.LongInstanceNameLongInstanceNameLongInstanceNameLongInstanceNameLongInstanceNameLongInstanceNameLongInstanceNameLongInstanceNameLongInstanceNameLongInstanceName@LONGTESTNAMELONGTESTNAMELONGTESTNAMELONGTESTNAMELONGTESTNAMELONGTESTNAMELONGTESTNAGAV';
    ShortTestMessage : T_MaxString := 'Very short message';

    // @Test-Result-Expected
    TestInstancePathNameWith252CharsExpectedResult : T_MaxString := 'PRG_TEST.LongInstanceNameLongInstanceNameLongInstanceNameLongInstanceNameLongInstanceNameLongInstanceNameLongInstanceNameLongInstanceNameLongInstanceNameLongInstanceName@LONGTESTNAMELONGTESTNAMELONGTESTNAMELONGTESTNAMELONGTESTNAMELO...TestName too long';
    ShortTestMessageExpectedResult : T_MaxString := '';

    // @Test-Result
    TestInstancePathNameWith252CharsResult : T_MaxString;
    ShortTestMessageResult : T_MaxString;
END_VAR
TEST('TestInstancePath255CharsExpectTooLongTestInstancePath');

AdjustAssertFailureMessageToMaxAllowedLength(TestInstancePath := TestInstancePathNameWith255Chars,
                                             TestMessage := ShortTestMessage,
                                             TestInstancePathProcessed => TestInstancePathNameWith252CharsResult,
                                             TestMessageProcessed => ShortTestMessageResult);

AssertEquals_STRING(Expected := TestInstancePathNameWith252CharsExpectedResult,
                    Actual := TestInstancePathNameWith252CharsResult,
                    'Test instance path not correct');

AssertEquals_STRING(Expected := ShortTestMessageExpectedResult,
                    Actual := ShortTestMessageResult,
                    'Test message not correct');

TEST_FINISHED();
END_METHOD

END_FUNCTION_BLOCK

// ---- Test/FB_EmptyTestSuite.TcPOU
(* This is an empty testsuite with no test cases, so that we can verify that the system still prints the
   test results. *)
FUNCTION_BLOCK FB_EmptyTestSuite EXTENDS TcUnit.FB_TestSuite
VAR
END_VAR

END_FUNCTION_BLOCK

// ---- Test/FB_CheckIfSpecificTestIsFinished.TcPOU
// Verifies that the function IS_TEST_FINISHED('Name') works as intended.
FUNCTION_BLOCK FB_CheckIfSpecificTestIsFinished EXTENDS TcUnit.FB_TestSuite

CheckBeforeAndAfterFinishing();

METHOD CheckBeforeAndAfterFinishing
TEST('CheckBeforeAndAfterFinishing');

AssertEquals_BOOL(Expected := FALSE,
                  Actual := IS_TEST_FINISHED('CheckBeforeAndAfterFinishing'),
                  Message:='Values differ before finishing');

TEST_FINISHED();

AssertEquals_BOOL(Expected := TRUE,
                  Actual := IS_TEST_FINISHED('CheckBeforeAndAfterFinishing'),
                  Message:='Values differ after finishing');
END_METHOD

END_FUNCTION_BLOCK

// ---- Test/FB_WriteProtectedFunctions.TcPOU
// This testsuite tests the WRITE_PROTECTED_* helper functions.
FUNCTION_BLOCK FB_WriteProtectedFunctions EXTENDS TcUnit.FB_TestSuite

Test_WRITE_PROTECTED_BOOL();
Test_WRITE_PROTECTED_BYTE();
Test_WRITE_PROTECTED_DATE();
Test_WRITE_PROTECTED_DATE_AND_TIME();
Test_WRITE_PROTECTED_DINT();
Test_WRITE_PROTECTED_DWORD();
Test_WRITE_PROTECTED_INT();
TEST_WRITE_PROTECTED_LINT();
Test_WRITE_PROTECTED_LREAL();
Test_WRITE_PROTECTED_LWORD();
Test_WRITE_PROTECTED_REAL();
Test_WRITE_PROTECTED_SINT();
Test_WRITE_PROTECTED_STRING();
Test_WRITE_PROTECTED_TIME();
Test_WRITE_PROTECTED_TIME_OF_DAY();
Test_WRITE_PROTECTED_UDINT();
Test_WRITE_PROTECTED_UINT();
Test_WRITE_PROTECTED_USINT();
Test_WRITE_PROTECTED_ULINT();
Test_WRITE_PROTECTED_WORD();
Test_WRITE_PROTECTED_WSTRING();

METHOD Test_WRITE_PROTECTED_BOOL
VAR
    ProtectedVariables : FB_ProtectedVariables;
END_VAR
TEST('Test_WRITE_PROTECTED_BOOL');

WRITE_PROTECTED_BOOL(ADR(ProtectedVariables.InputBOOL), TRUE);
AssertEquals_BOOL(TRUE, ProtectedVariables.InputBOOL, 'Overwriting protected InputBOOL');

WRITE_PROTECTED_BOOL(ADR(ProtectedVariables.VarBOOL), TRUE);
AssertEquals_BOOL(TRUE, ProtectedVariables.VarBOOL, 'Overwriting protected VarBOOL');

TEST_FINISHED();
END_METHOD

METHOD Test_WRITE_PROTECTED_BYTE
VAR
    ProtectedVariables : FB_ProtectedVariables;
END_VAR
TEST('Test_WRITE_PROTECTED_BYTE');

WRITE_PROTECTED_BYTE(ADR(ProtectedVariables.InputBYTE), 1);
AssertEquals_BYTE(1, ProtectedVariables.InputBYTE, 'Overwriting protected InputBYTE');

WRITE_PROTECTED_BYTE(ADR(ProtectedVariables.VarBYTE), 1);
AssertEquals_BYTE(1, ProtectedVariables.VarBYTE, 'Overwriting protected VarBYTE');

TEST_FINISHED();
END_METHOD

METHOD Test_WRITE_PROTECTED_DATE
VAR
    ProtectedVariables : FB_ProtectedVariables;
END_VAR
TEST('Test_WRITE_PROTECTED_DATE');

WRITE_PROTECTED_DATE(ADR(ProtectedVariables.InputDATE), D#2000-01-01);
AssertEquals_DATE(D#2000-01-01, ProtectedVariables.InputDATE, 'Overwriting protected InputDATE');

WRITE_PROTECTED_DATE(ADR(ProtectedVariables.VarDATE), D#2000-01-01);
AssertEquals_DATE(D#2000-01-01, ProtectedVariables.VarDATE, 'Overwriting protected VarDATE');

TEST_FINISHED();
END_METHOD

METHOD Test_WRITE_PROTECTED_DATE_AND_TIME
VAR
    ProtectedVariables : FB_ProtectedVariables;
END_VAR
TEST('Test_WRITE_PROTECTED_DATE_AND_TIME');

WRITE_PROTECTED_DATE_AND_TIME(ADR(ProtectedVariables.InputDATE_AND_TIME), DT#2000-01-01-00:00);
AssertEquals_DATE_AND_TIME(DT#2000-01-01-00:00, ProtectedVariables.InputDATE_AND_TIME, 'Overwriting protected InputDATE_AND_TIME');

WRITE_PROTECTED_DATE_AND_TIME(ADR(ProtectedVariables.VarDATE_AND_TIME), DT#2000-01-01-00:00);
AssertEquals_DATE_AND_TIME(DT#2000-01-01-00:00, ProtectedVariables.VarDATE_AND_TIME, 'Overwriting protected VarDATE_AND_TIME');

TEST_FINISHED();
END_METHOD

METHOD Test_WRITE_PROTECTED_DINT
VAR
    ProtectedVariables : FB_ProtectedVariables;
END_VAR
TEST('Test_WRITE_PROTECTED_DINT');

WRITE_PROTECTED_DINT(ADR(ProtectedVariables.InputDINT), 1);
AssertEquals_DINT(1, ProtectedVariables.InputDINT, 'Overwriting protected InputDINT');

WRITE_PROTECTED_DINT(ADR(ProtectedVariables.VarDINT), 1);
AssertEquals_DINT(1, ProtectedVariables.VarDINT, 'Overwriting protected VarDINT');

TEST_FINISHED();
END_METHOD

METHOD Test_WRITE_PROTECTED_DWORD
VAR
    ProtectedVariables : FB_ProtectedVariables;
END_VAR
TEST('Test_WRITE_PROTECTED_DWORD');

WRITE_PROTECTED_DWORD(ADR(ProtectedVariables.InputDWORD), 1);
AssertEquals_DWORD(1, ProtectedVariables.InputDWORD, 'Overwriting protected InputDWORD');

WRITE_PROTECTED_DWORD(ADR(ProtectedVariables.VarDWORD), 1);
AssertEquals_DWORD(1, ProtectedVariables.VarDWORD, 'Overwriting protected VarDWORD');

TEST_FINISHED();
END_METHOD

METHOD Test_WRITE_PROTECTED_INT
VAR
    ProtectedVariables : FB_ProtectedVariables;
END_VAR
TEST('Test_WRITE_PROTECTED_INT');

WRITE_PROTECTED_INT(ADR(ProtectedVariables.InputINT), 1);
AssertEquals_INT(1, ProtectedVariables.InputINT, 'Overwriting protected InputINT');

WRITE_PROTECTED_INT(ADR(ProtectedVariables.VarINT), 1);
AssertEquals_INT(1, ProtectedVariables.VarINT, 'Overwriting protected VarINT');

TEST_FINISHED();
END_METHOD

METHOD Test_WRITE_PROTECTED_LINT
VAR
    ProtectedVariables : FB_ProtectedVariables;
END_VAR
TEST('Test_WRITE_PROTECTED_LINT');

WRITE_PROTECTED_LINT(ADR(ProtectedVariables.InputLINT), 5);
AssertEquals_LINT(5, ProtectedVariables.InputLINT, 'Overwriting protected InputLINT');

WRITE_PROTECTED_LINT(ADR(ProtectedVariables.VarLINT), 5);
AssertEquals_LINT(5, ProtectedVariables.VarLINT, 'Overwriting protected VarLINT');

TEST_FINISHED();
END_METHOD

METHOD Test_WRITE_PROTECTED_LREAL
VAR
    ProtectedVariables : FB_ProtectedVariables;
END_VAR
TEST('Test_WRITE_PROTECTED_LREAL');

WRITE_PROTECTED_LREAL(ADR(ProtectedVariables.InputLREAL), 1);
AssertEquals_LREAL(1, ProtectedVariables.InputLREAL, 0, 'Overwriting protected InputLREAL');

WRITE_PROTECTED_LREAL(ADR(ProtectedVariables.VarLREAL), 1);
AssertEquals_LREAL(1, ProtectedVariables.VarLREAL, 0, 'Overwriting protected VarLREAL');

TEST_FINISHED();
END_METHOD

METHOD Test_WRITE_PROTECTED_LWORD
VAR
    ProtectedVariables : FB_ProtectedVariables;
END_VAR
TEST('Test_WRITE_PROTECTED_LWORD');

WRITE_PROTECTED_LWORD(ADR(ProtectedVariables.InputLWORD), 4);
AssertEquals_LWORD(4, ProtectedVariables.InputLWORD, 'Overwriting protected InputLWORD');

WRITE_PROTECTED_LWORD(ADR(ProtectedVariables.VarLWORD), 4);
AssertEquals_LWORD(4, ProtectedVariables.VarLWORD, 'Overwriting protected VarLWORD');

TEST_FINISHED();
END_METHOD

METHOD Test_WRITE_PROTECTED_REAL
VAR
    ProtectedVariables : FB_ProtectedVariables;
END_VAR
TEST('Test_WRITE_PROTECTED_REAL');

WRITE_PROTECTED_REAL(ADR(ProtectedVariables.InputREAL), 1);
AssertEquals_REAL(1, ProtectedVariables.InputREAL, 0, 'Overwriting protected InputREAL');

WRITE_PROTECTED_REAL(ADR(ProtectedVariables.VarREAL), 1);
AssertEquals_REAL(1, ProtectedVariables.VarREAL, 0, 'Overwriting protected VarREAL');

TEST_FINISHED();
END_METHOD

METHOD Test_WRITE_PROTECTED_SINT
VAR
    ProtectedVariables : FB_ProtectedVariables;
END_VAR
TEST('Test_WRITE_PROTECTED_SINT');

WRITE_PROTECTED_SINT(ADR(ProtectedVariables.InputSINT), 1);
AssertEquals_SINT(1, ProtectedVariables.InputSINT, 'Overwriting protected InputSINT');

WRITE_PROTECTED_SINT(ADR(ProtectedVariables.VarSINT), 1);
AssertEquals_SINT(1, ProtectedVariables.VarSINT, 'Overwriting protected VarSINT');

TEST_FINISHED();
END_METHOD

METHOD Test_WRITE_PROTECTED_STRING
VAR
    ProtectedVariables : FB_ProtectedVariables;
END_VAR
TEST('Test_WRITE_PROTECTED_STRING');

WRITE_PROTECTED_STRING(ADR(ProtectedVariables.InputSTRING), 'words');
AssertEquals_STRING('words', ProtectedVariables.InputSTRING, 'Overwriting protected InputSTRING');

WRITE_PROTECTED_STRING(ADR(ProtectedVariables.VarSTRING), 'words');
AssertEquals_STRING('words', ProtectedVariables.VarSTRING, 'Overwriting protected VarSTRING');

TEST_FINISHED();
END_METHOD

METHOD Test_WRITE_PROTECTED_TIME
VAR
    ProtectedVariables : FB_ProtectedVariables;
END_VAR
TEST('Test_WRITE_PROTECTED_TIME');

WRITE_PROTECTED_TIME(ADR(ProtectedVariables.InputTIME), T#1S);
AssertEquals_TIME(T#1S, ProtectedVariables.InputTIME, 'Overwriting protected InputTIME');

WRITE_PROTECTED_TIME(ADR(ProtectedVariables.VarTIME), T#1S);
AssertEquals_TIME(T#1S, ProtectedVariables.VarTIME, 'Overwriting protected VarTIME');

TEST_FINISHED();
END_METHOD

METHOD Test_WRITE_PROTECTED_TIME_OF_DAY
VAR
    ProtectedVariables : FB_ProtectedVariables;
END_VAR
TEST('Test_WRITE_PROTECTED_TIME_OF_DAY');

WRITE_PROTECTED_TIME_OF_DAY(ADR(ProtectedVariables.InputTIME_OF_DAY), TOD#11:11);
AssertEquals_TIME_OF_DAY(TOD#11:11, ProtectedVariables.InputTIME_OF_DAY, 'Overwriting protected InputTIME_OF_DAY');

WRITE_PROTECTED_TIME_OF_DAY(ADR(ProtectedVariables.VarTIME_OF_DAY), TOD#11:11);
AssertEquals_TIME_OF_DAY(TOD#11:11, ProtectedVariables.VarTIME_OF_DAY, 'Overwriting protected VarTIME_OF_DAY');

TEST_FINISHED();
END_METHOD

METHOD Test_WRITE_PROTECTED_UDINT
VAR
    ProtectedVariables : FB_ProtectedVariables;
END_VAR
TEST('Test_WRITE_PROTECTED_UDINT');

WRITE_PROTECTED_UDINT(ADR(ProtectedVariables.InputUDINT), 1);
AssertEquals_UDINT(1, ProtectedVariables.InputUDINT, 'Overwriting protected InputUDINT');

WRITE_PROTECTED_UDINT(ADR(ProtectedVariables.VarUDINT), 1);
AssertEquals_UDINT(1, ProtectedVariables.VarUDINT, 'Overwriting protected VarUDINT');

TEST_FINISHED();
END_METHOD

METHOD Test_WRITE_PROTECTED_UINT
VAR
    ProtectedVariables : FB_ProtectedVariables;
END_VAR
TEST('Test_WRITE_PROTECTED_UINT');

WRITE_PROTECTED_UINT(ADR(ProtectedVariables.InputUINT), 1);
AssertEquals_UINT(1, ProtectedVariables.InputUINT, 'Overwriting protected InputUINT');

WRITE_PROTECTED_UINT(ADR(ProtectedVariables.VarUINT), 1);
AssertEquals_UINT(1, ProtectedVariables.VarUINT, 'Overwriting protected VarUINT');

TEST_FINISHED();
END_METHOD

METHOD Test_WRITE_PROTECTED_ULINT
VAR
    ProtectedVariables : FB_ProtectedVariables;
END_VAR
TEST('Test_WRITE_PROTECTED_ULINT');

WRITE_PROTECTED_ULINT(ADR(ProtectedVariables.InputULINT), 8);
AssertEquals_ULINT(8, ProtectedVariables.InputULINT, 'Overwriting protected InputULINT');

WRITE_PROTECTED_ULINT(ADR(ProtectedVariables.VarULINT), 8);
AssertEquals_ULINT(8, ProtectedVariables.VarULINT, 'Overwriting protected VarULINT');

TEST_FINISHED();
END_METHOD

METHOD Test_WRITE_PROTECTED_USINT
VAR
    ProtectedVariables : FB_ProtectedVariables;
END_VAR
TEST('Test_WRITE_PROTECTED_USINT');

WRITE_PROTECTED_USINT(ADR(ProtectedVariables.InputUSINT), 1);
AssertEquals_USINT(1, ProtectedVariables.InputUSINT, 'Overwriting protected InputUSINT');

WRITE_PROTECTED_USINT(ADR(ProtectedVariables.VarUSINT), 1);
AssertEquals_USINT(1, ProtectedVariables.VarUSINT, 'Overwriting protected VarUSINT');

TEST_FINISHED();
END_METHOD

METHOD Test_WRITE_PROTECTED_WORD
VAR
    ProtectedVariables : FB_ProtectedVariables;
END_VAR
TEST('Test_WRITE_PROTECTED_WORD');

WRITE_PROTECTED_WORD(ADR(ProtectedVariables.InputWORD), 1);
AssertEquals_WORD(1, ProtectedVariables.InputWORD, 'Overwriting protected InputWORD');

WRITE_PROTECTED_WORD(ADR(ProtectedVariables.VarWORD), 1);
AssertEquals_WORD(1, ProtectedVariables.VarWORD, 'Overwriting protected VarWORD');

TEST_FINISHED();
END_METHOD

METHOD Test_WRITE_PROTECTED_WSTRING
VAR
    ProtectedVariables : FB_ProtectedVariables;
END_VAR
TEST('Test_WRITE_PROTECTED_WSTRING');

WRITE_PROTECTED_WSTRING(ADR(ProtectedVariables.InputWSTRING), "ŢŶǮ");
AssertEquals_WSTRING("ŢŶǮ", ProtectedVariables.InputWSTRING, 'Overwriting protected InputWSTRING');

WRITE_PROTECTED_WSTRING(ADR(ProtectedVariables.VarWSTRING), "ŢŶǮ");
AssertEquals_WSTRING("ŢŶǮ", ProtectedVariables.VarWSTRING, 'Overwriting protected VarWSTRING');

TEST_FINISHED();
END_METHOD

END_FUNCTION_BLOCK

// ---- POUs/FB_ProtectedVariables.TcPOU
(*
    Contains different types of "protected" variables that you could not normally write to in
    production PLC code, but would need to overwrite for testing purposes. Used for testing the
    WRITE_PROTECTED_* functions, but this FB doesn't contain any tests itself.
*)
FUNCTION_BLOCK FB_ProtectedVariables
VAR_INPUT
    InputBOOL AT %I* : BOOL;
    InputBYTE AT %I* : BYTE;
    InputDATE AT %I* : DATE;
    InputDATE_AND_TIME AT %I* : DATE_AND_TIME;
    InputDINT AT %I* : DINT;
    InputDWORD AT %I* : DWORD;
    InputINT AT %I* : INT;
    InputLINT AT %I* : LINT;
    InputLREAL AT %I* : LREAL;
    InputLWORD AT %I* : LWORD;
    InputREAL AT %I* : REAL;
    InputSINT AT %I* : SINT;
    InputSTRING AT %I* : STRING;
    InputTIME AT %I* : TIME;
    InputTIME_OF_DAY AT %I* : TIME_OF_DAY;
    InputUDINT AT %I* : UDINT;
    InputUINT AT %I* : UINT;
    InputULINT AT %I* : ULINT;
    InputUSINT AT %I* : USINT;
    InputWORD AT %I* : WORD;
    InputWSTRING AT %I* : WSTRING;
END_VAR
VAR
    VarBOOL : BOOL;
    VarBYTE : BYTE;
    VarDATE : DATE;
    VarDATE_AND_TIME : DATE_AND_TIME;
    VarDINT : DINT;
    VarDWORD : DWORD;
    VarINT : INT;
    VarLINT : LINT;
    VarLREAL : LREAL;
    VarLWORD : LWORD;
    VarREAL : REAL;
    VarSINT : SINT;
    VarSTRING : STRING;
    VarTIME : TIME;
    VarTIME_OF_DAY : TIME_OF_DAY;
    VarUDINT : UDINT;
    VarUINT : UINT;
    VarULINT : ULINT;
    VarUSINT : USINT;
    VarWORD : WORD;
    VarWSTRING : WSTRING;
END_VAR

END_FUNCTION_BLOCK

// ---- Test/FB_TestNumberOfAssertionsCalculation.TcPOU
// This testsuite verifies that the number of assertions for every testcase is correctly calculated
FUNCTION_BLOCK FB_TestNumberOfAssertionsCalculation EXTENDS TcUnit.FB_TestSuite

TestMixed33SuccessulAnd9FailedAssertions();
TestWith43SuccessfulAssertions();
TestWith44FailedAssertions();
TestWith45SuccessfulArrayAssertions();
TestWith46FailedArrayAssertions();

METHOD PRIVATE TestMixed33SuccessulAnd9FailedAssertions
VAR
    // Successful
    aAny : INT := 5;
    bAny : INT := 5;

    // Successful
    aBool : BOOL := TRUE;
    bBool : BOOL := TRUE;

    // Failed
    aDint : ARRAY[2..7] OF DINT := [64, 98, 2147483647, -2147483648, 0, -63987538];
    bDint : ARRAY[1..5] OF DINT := [64, 98, 2147483647, -2147483648, 0];

    // Failed
    aDword : ARRAY[2..3] OF DWORD := [16#6789ABCD, 16#EF012345];
    bDword : ARRAY[1..2] OF DWORD := [16#6789ABCD, 16#EF012343];

    // Successful
    aInt : ARRAY[-5..1] OF INT := [64, 98, -32768, 32767, 5478, -378, 42];
    bInt : ARRAY[1..7] OF INT := [64, 98, -32768, 32767, 5478, -378, 42];

    // Successful
    aLint : ARRAY[-1..0] OF LINT := [9_223_372_036_854_775_807, -9_223_372_036_854_775_808];
    bLint : ARRAY[4..5] OF LINT := [9_223_372_036_854_775_807, -9_223_372_036_854_775_808];

    // Failed
    aLreal : LREAL := 1234564.89;
    bLreal : LREAL := 1234567.76;

    // Failed
    aLtime : LTIME := LTIME#213503D23H33M33S709MS551US615NS;
    bLtime : LTIME := LTIME#213503D23H34M33S709MS551US615NS;

    // Failed
    aLrealArray : ARRAY[-5..1] OF LREAL := [64.0, 97.1, -32768.2, 32767.3, 5478.4, -378.5, 42.6];
    bLrealArray : ARRAY[1..7] OF LREAL := [64.0001, 98.0999, -32768.1995, 32767.3001, 5478.4002, -378.5003, 42.6001];

    // Failed
    aLreal2d : ARRAY[-5..-3,-1..0] OF LREAL := [64.0, 98.1, -32768.2, 32767.3, 5478.4, -378.5];
    bLreal2d : ARRAY[1..3,0..1] OF LREAL := [63.0001, 98.0999, -32768.1995, 32767.3001, 5478.4002, -378.5003];

    // Successful
    aLword : LWORD := 16#0123456789ABCDEF;
    bLword : LWORD := 16#0123456789ABCDEF;

    // Successful
    aSint : SINT := -128;
    bSint : SINT := -128;

    // Successful
    aUdint : ARRAY[1..3] OF UDINT := [0, 4294967295, 5000];
    bUdint : ARRAY[1..3] OF UDINT := [0, 4294967295, 5000];

    // Successful
    aUint : ARRAY[0..4] OF UINT := [0, 65535, 2000, 34123, 59];
    bUint : ARRAY[0..4] OF UINT := [0, 65535, 2000, 34123, 59];

    // Failed
    aUlint : ULINT := 45683838382;
    bUlint : ULINT := 45683838383;

    // Failed
    aUsint : USINT := 4;
    bUsint : USINT := 5;

    // Failed
    aWord : ARRAY[1..5] OF WORD := [16#AAAA, 16#BBBF, 16#CCCC, 16#DDDD, 16#EEEE];
    bWord : ARRAY[1..5] OF WORD := [16#AAAA, 16#BBBB, 16#CCCC, 16#DDDD, 16#EEEE];

    // Successful
    aSintDummy1 : SINT := 1;
    bSintDummy1 : SINT := 1;

    // Successful
    aSintDummy2 : SINT := 2;
    bSintDummy2 : SINT := 2;

    // Successful
    aSintDummy3 : SINT := 3;
    bSintDummy3 : SINT := 3;

    // Successful
    aSintDummy4 : SINT := 4;
    bSintDummy4 : SINT := 4;

    // Successful
    aSintDummy5 : SINT := 5;
    bSintDummy5 : SINT := 5;

    // Successful
    aSintDummy6 : SINT := 6;
    bSintDummy6 : SINT := 6;

    // Successful
    aSintDummy7 : SINT := 7;
    bSintDummy7 : SINT := 7;

    // Successful
    aSintDummy8 : SINT := 8;
    bSintDummy8 : SINT := 8;

    // Successful
    aSintDummy9 : SINT := 9;
    bSintDummy9 : SINT := 9;

    // Successful
    aSintDummy10 : SINT := 10;
    bSintDummy10 : SINT := 10;

    // Successful
    aSintDummy11 : SINT := 11;
    bSintDummy11 : SINT := 11;

    // Successful
    aSintDummy12 : SINT := 12;
    bSintDummy12 : SINT := 12;

    // Successful
    aSintDummy13 : SINT := 13;
    bSintDummy13 : SINT := 13;

    // Successful
    aSintDummy14 : SINT := 14;
    bSintDummy14 : SINT := 14;

    // Successful
    aSintDummy15 : SINT := 15;
    bSintDummy15 : SINT := 15;

    // Successful
    aSintDummy16 : SINT := 16;
    bSintDummy16 : SINT := 16;

    // Successful
    aSintDummy17 : SINT := 17;
    bSintDummy17 : SINT := 17;

    // Successful
    aSintDummy18 : SINT := 18;
    bSintDummy18 : SINT := 18;

    // Successful
    aSintDummy19 : SINT := 19;
    bSintDummy19 : SINT := 19;

    // Successful
    aSintDummy20 : SINT := 20;
    bSintDummy20 : SINT := 20;

    // Successful
    aSintDummy21 : SINT := 21;
    bSintDummy21 : SINT := 21;

    // Successful
    aSintDummy22 : SINT := 22;
    bSintDummy22 : SINT := 22;

    // Successful
    aSintDummy23 : SINT := 23;
    bSintDummy23 : SINT := 23;

    // Successful
    aSintDummy24 : SINT := 24;
    bSintDummy24 : SINT := 24;

    // Successful
    aSintDummy25 : SINT := 25;
    bSintDummy25 : SINT := 25;
END_VAR
TEST('TestMixed33SuccessulAnd9FailedAssertions');

AssertEquals(Expected := aAny,
             Actual := bAny,
             Message := 'Values differ');

AssertEquals_BOOL(Expected := aBool,
                  Actual := bBool,
                  Message := 'Values differ');

AssertArrayEquals_DINT(Expecteds := aDint,
                       Actuals := bDint,
                       Message := 'Arrays differ');

AssertArrayEquals_DWORD(Expecteds := aDword,
                        Actuals := bDword,
                        Message := 'Arrays differ');

AssertArrayEquals_INT(Expecteds := aInt,
                      Actuals := bInt,
                      Message := 'Arrays differ');

AssertArrayEquals_LINT(Expecteds := aLint,
                      Actuals := bLint,
                      Message := 'Arrays differ');

AssertEquals_LREAL(Expected := aLreal,
                   Actual := bLreal,
                   Delta := 0.2,
                   Message := 'Values differ');

AssertEquals_LTIME(Expected := aLtime,
                   Actual := bLtime,
                   Message := 'Values differ');

AssertArrayEquals_LREAL(Expecteds := aLrealArray,
                        Actuals := bLrealArray,
                        Delta := 0.01,
                        Message := 'Arrays differ');

AssertArray2dEquals_LREAL(Expecteds := aLreal2d,
                          Actuals := bLreal2d,
                          Delta := 0.01,
                          Message := 'Arrays differ');

AssertEquals_LWORD(Expected := aLword,
                   Actual := bLword,
                   Message := 'Values differ');

AssertEquals_SINT(Expected := aSint,
                  Actual := bSint,
                  Message := 'Values differ');

AssertArrayEquals_UDINT(Expecteds := aUdint,
                        Actuals := bUdint,
                        Message := 'Arrays differ');

AssertArrayEquals_UINT(Expecteds := aUint,
                       Actuals := bUint,
                       Message := 'Arrays differ');

AssertEquals_ULINT(Expected := aUlint,
                   Actual := bUlint,
                   Message := 'Values differ');

AssertEquals_USINT(Expected := aUsint,
                   Actual := bUsint,
                   Message := 'Values differ');

AssertArrayEquals_WORD(Expecteds := aWord,
                       Actuals := bWord,
                       Message := 'Arrays differ');

AssertEquals_SINT(Expected := aSintDummy1,
                  Actual := bSintDummy1,
                  Message := 'Values differ');

AssertEquals_SINT(Expected := aSintDummy2,
                  Actual := bSintDummy2,
                  Message := 'Values differ');

AssertEquals_SINT(Expected := aSintDummy3,
                  Actual := bSintDummy3,
                  Message := 'Values differ');

AssertEquals_SINT(Expected := aSintDummy4,
                  Actual := bSintDummy4,
                  Message := 'Values differ');

AssertEquals_SINT(Expected := aSintDummy5,
                  Actual := bSintDummy5,
                  Message := 'Values differ');

AssertEquals_SINT(Expected := aSintDummy6,
                  Actual := bSintDummy6,
                  Message := 'Values differ');

AssertEquals_SINT(Expected := aSintDummy7,
                  Actual := bSintDummy7,
                  Message := 'Values differ');

AssertEquals_SINT(Expected := aSintDummy8,
                  Actual := bSintDummy8,
                  Message := 'Values differ');

AssertEquals_SINT(Expected := aSintDummy9,
                  Actual := bSintDummy9,
                  Message := 'Values differ');

AssertEquals_SINT(Expected := aSintDummy10,
                  Actual := bSintDummy10,
                  Message := 'Values differ');

AssertEquals_SINT(Expected := aSintDummy11,
                  Actual := bSintDummy11,
                  Message := 'Values differ');

AssertEquals_SINT(Expected := aSintDummy12,
                  Actual := bSintDummy12,
                  Message := 'Values differ');

AssertEquals_SINT(Expected := aSintDummy13,
                  Actual := bSintDummy13,
                  Message := 'Values differ');

AssertEquals_SINT(Expected := aSintDummy14,
                  Actual := bSintDummy14,
                  Message := 'Values differ');

AssertEquals_SINT(Expected := aSintDummy15,
                  Actual := bSintDummy15,
                  Message := 'Values differ');

AssertEquals_SINT(Expected := aSintDummy16,
                  Actual := bSintDummy16,
                  Message := 'Values differ');

AssertEquals_SINT(Expected := aSintDummy17,
                  Actual := bSintDummy17,
                  Message := 'Values differ');

AssertEquals_SINT(Expected := aSintDummy18,
                  Actual := bSintDummy18,
                  Message := 'Values differ');

AssertEquals_SINT(Expected := aSintDummy19,
                  Actual := bSintDummy19,
                  Message := 'Values differ');

AssertEquals_SINT(Expected := aSintDummy20,
                  Actual := bSintDummy20,
                  Message := 'Values differ');

AssertEquals_SINT(Expected := aSintDummy21,
                  Actual := bSintDummy21,
                  Message := 'Values differ');

AssertEquals_SINT(Expected := aSintDummy22,
                  Actual := bSintDummy22,
                  Message := 'Values differ');

AssertEquals_SINT(Expected := aSintDummy23,
                  Actual := bSintDummy23,
                  Message := 'Values differ');

AssertEquals_SINT(Expected := aSintDummy24,
                  Actual := bSintDummy24,
                  Message := 'Values differ');

AssertEquals_SINT(Expected := aSintDummy25,
                  Actual := bSintDummy25,
                  Message := 'Values differ');

TEST_FINISHED();
END_METHOD

METHOD PRIVATE TestWith43SuccessfulAssertions
VAR
    aAny : INT := 5;
    bAny : INT := 5;

    aBool : BOOL := TRUE;
    bBool : BOOL := TRUE;

    aByte : BYTE := 16#CD;
    bByte : BYTE := 16#CD;

    aDateAndTime : DATE_AND_TIME := DATE_AND_TIME#2019-01-20-13:54:30;
    bDateAndTime : DATE_AND_TIME := DATE_AND_TIME#2019-01-20-13:54:30;

    aDate : DATE := DATE#1996-05-06;
    bDate : DATE := DATE#1996-05-06;

    aDint : DINT := -80000;
    bDint : DINT := -80000;

    aDword : DWORD := 16#7890ABCD;
    bDword : DWORD := 16#7890ABCD;


    aInt : INT := -12345;
    bInt : INT := -12345;

    aLint : LINT := -123456789;
    bLint : LINT := -123456789;

    aLreal : LREAL := 1234567.89;
    bLreal : LREAL := 1234567.76;

    aLtime : LTIME := LTIME#213503D23H34M33S709MS551US615NS;
    bLtime : LTIME := LTIME#213503D23H34M33S709MS551US615NS;

    aLword : LWORD := 16#0123456789ABCDEF;
    bLword : LWORD := 16#0123456789ABCDEF;

    aReal : REAL := 1234.5;
    bReal : REAL := 1234.4;

    aSint : SINT := -128;
    bSint : SINT := -128;

    aString : STRING := 'Hello there';
    bString : STRING := 'Hello there';

    aTime : TIME := T#11H34M13S244MS;
    bTime : TIME := T#11H34M13S244MS;

    aTimeOfDay : TIME_OF_DAY := TIME_OF_DAY#06:21:11.492;
    bTimeOfDay : TIME_OF_DAY := TIME_OF_DAY#06:21:11.492;

    aUdint : UDINT := 21845123;
    bUdint : UDINT := 21845123;

    aUint : UINT := 65535;
    bUint : UINT := 65535;

    aUlint : ULINT := 45683838383;
    bUlint : ULINT := 45683838383;

    aUsint : USINT := 5;
    bUsint : USINT := 5;

    aWord : WORD := 16#ABCD;
    bWord : WORD := 16#ABCD;

    aSintDummy1 : SINT := 1;
    bSintDummy1 : SINT := 1;

    aSintDummy2 : SINT := 2;
    bSintDummy2 : SINT := 2;

    aSintDummy3 : SINT := 3;
    bSintDummy3 : SINT := 3;

    aSintDummy4 : SINT := 4;
    bSintDummy4 : SINT := 4;

    aSintDummy5 : SINT := 5;
    bSintDummy5 : SINT := 5;

    aSintDummy6 : SINT := 6;
    bSintDummy6 : SINT := 6;

    aSintDummy7 : SINT := 7;
    bSintDummy7 : SINT := 7;

    aSintDummy8 : SINT := 8;
    bSintDummy8 : SINT := 8;

    aSintDummy9 : SINT := 9;
    bSintDummy9 : SINT := 9;

    aSintDummy10 : SINT := 10;
    bSintDummy10 : SINT := 10;

    aSintDummy11 : SINT := 11;
    bSintDummy11 : SINT := 11;

    aSintDummy12 : SINT := 12;
    bSintDummy12 : SINT := 12;

    aSintDummy13 : SINT := 13;
    bSintDummy13 : SINT := 13;

    aSintDummy14 : SINT := 14;
    bSintDummy14 : SINT := 14;

    aSintDummy15 : SINT := 15;
    bSintDummy15 : SINT := 15;

    aSintDummy16 : SINT := 16;
    bSintDummy16 : SINT := 16;

    aSintDummy17 : SINT := 17;
    bSintDummy17 : SINT := 17;

    aSintDummy18 : SINT := 18;
    bSintDummy18 : SINT := 18;

    aSintDummy19 : SINT := 19;
    bSintDummy19 : SINT := 19;

    aSintDummy20 : SINT := 20;
    bSintDummy20 : SINT := 20;

    aSintDummy21 : SINT := 21;
    bSintDummy21 : SINT := 21;
END_VAR
TEST('TestWith22SuccessfulAssertions');

AssertEquals(Expected := aAny,
             Actual := bAny,
             Message := 'Values differ');

AssertEquals_BOOL(Expected := aBool,
                  Actual := bBool,
                  Message := 'Values differ');

AssertEquals_BYTE(Expected := aByte,
                  Actual := bByte,
                  Message := 'Values differ');

AssertEquals_DATE_AND_TIME(Expected := aDateAndTime,
                           Actual := bDateAndTime,
                           Message := 'Values differ');

AssertEquals_DATE(Expected := aDate,
                  Actual := bDate,
                  Message := 'Values differ');

AssertEquals_DINT(Expected := aDint,
                  Actual := bDint,
                  Message := 'Values differ');

AssertEquals_DWORD(Expected := aDword,
                   Actual := bDword,
                   Message := 'Values differ');

AssertEquals_INT(Expected := aInt,
                 Actual := bInt,
                 Message := 'Values differ');

AssertEquals_LINT(Expected := aLint,
                  Actual := bLint,
                  Message := 'Values differ');

AssertEquals_LREAL(Expected := aLreal,
                   Actual := bLreal,
                   Delta := 0.2,
                   Message := 'Values differ');

AssertEquals_LTIME(Expected := aLtime,
                   Actual := bLtime,
                   Message := 'Values differ');

AssertEquals_LWORD(Expected := aLword,
                   Actual := bLword,
                   Message := 'Values differ');

AssertEquals_REAL(Expected := aReal,
                  Actual := bReal,
                  Delta := 0.1,
                  Message := 'Values differ');

AssertEquals_SINT(Expected := aSint,
                  Actual := bSint,
                  Message := 'Values differ');

AssertEquals_STRING(Expected := aString,
                    Actual := bString,
                    Message := 'Values differ');

AssertEquals_TIME(Expected := aTime,
                  Actual := bTime,
                  Message := 'Values differ');

AssertEquals_TIME_OF_DAY(Expected := aTimeOfDay,
                         Actual := bTimeOfDay,
                         Message := 'Values differ');

AssertEquals_UDINT(Expected := aUdint,
                   Actual := bUdint,
                   Message := 'Values differ');

AssertEquals_UINT(Expected := aUint,
                  Actual := bUint,
                  Message := 'Values differ');

AssertEquals_ULINT(Expected := aUlint,
                   Actual := bUlint,
                   Message := 'Values differ');

AssertEquals_USINT(Expected := aUsint,
                   Actual := bUsint,
                   Message := 'Values differ');

AssertEquals_WORD(Expected := aWord,
                  Actual := bWord,
                  Message := 'Values differ');

AssertEquals_SINT(Expected := aSintDummy1,
                  Actual := bSintDummy1,
                  Message := 'Values differ');

AssertEquals_SINT(Expected := aSintDummy2,
                  Actual := bSintDummy2,
                  Message := 'Values differ');

AssertEquals_SINT(Expected := aSintDummy3,
                  Actual := bSintDummy3,
                  Message := 'Values differ');

AssertEquals_SINT(Expected := aSintDummy4,
                  Actual := bSintDummy4,
                  Message := 'Values differ');

AssertEquals_SINT(Expected := aSintDummy5,
                  Actual := bSintDummy5,
                  Message := 'Values differ');

AssertEquals_SINT(Expected := aSintDummy6,
                  Actual := bSintDummy6,
                  Message := 'Values differ');

AssertEquals_SINT(Expected := aSintDummy7,
                  Actual := bSintDummy7,
                  Message := 'Values differ');

AssertEquals_SINT(Expected := aSintDummy8,
                  Actual := bSintDummy8,
                  Message := 'Values differ');

AssertEquals_SINT(Expected := aSintDummy9,
                  Actual := bSintDummy9,
                  Message := 'Values differ');

AssertEquals_SINT(Expected := aSintDummy10,
                  Actual := bSintDummy10,
                  Message := 'Values differ');

AssertEquals_SINT(Expected := aSintDummy11,
                  Actual := bSintDummy11,
                  Message := 'Values differ');

AssertEquals_SINT(Expected := aSintDummy12,
                  Actual := bSintDummy12,
                  Message := 'Values differ');

AssertEquals_SINT(Expected := aSintDummy13,
                  Actual := bSintDummy13,
                  Message := 'Values differ');

AssertEquals_SINT(Expected := aSintDummy14,
                  Actual := bSintDummy14,
                  Message := 'Values differ');

AssertEquals_SINT(Expected := aSintDummy15,
                  Actual := bSintDummy15,
                  Message := 'Values differ');

AssertEquals_SINT(Expected := aSintDummy16,
                  Actual := bSintDummy16,
                  Message := 'Values differ');

AssertEquals_SINT(Expected := aSintDummy17,
                  Actual := bSintDummy17,
                  Message := 'Values differ');

AssertEquals_SINT(Expected := aSintDummy18,
                  Actual := bSintDummy18,
                  Message := 'Values differ');

AssertEquals_SINT(Expected := aSintDummy19,
                  Actual := bSintDummy19,
                  Message := 'Values differ');

AssertEquals_SINT(Expected := aSintDummy20,
                  Actual := bSintDummy20,
                  Message := 'Values differ');

AssertEquals_SINT(Expected := aSintDummy21,
                  Actual := bSintDummy21,
                  Message := 'Values differ');

TEST_FINISHED();
END_METHOD

METHOD PRIVATE TestWith44FailedAssertions
VAR
    aAny : INT := 5;
    bAny : INT := 4;

    aBool : BOOL := TRUE;
    bBool : BOOL := FALSE;

    aBool2 : BOOL := FALSE;
    bBool2 : BOOL := TRUE;

    aByte : BYTE := 16#AB;
    bByte : BYTE := 16#CD;

    aDateAndTime : DATE_AND_TIME := DATE_AND_TIME#2018-01-20-13:54:30;
    bDateAndTime : DATE_AND_TIME := DATE_AND_TIME#2019-01-20-13:54:30;

    aDate : DATE := DATE#1995-05-06;
    bDate : DATE := DATE#1996-05-06;

    aDint : DINT := -80001;
    bDint : DINT := -80000;

    aDword : DWORD := 16#7890ABDD;
    bDword : DWORD := 16#7890ABCD;

    aInt : INT := -12344;
    bInt : INT := -12345;

    aLint : LINT := -123456787;
    bLint : LINT := -123456789;

    aLreal : LREAL := 1234564.89;
    bLreal : LREAL := 1234567.76;

    aLtime : LTIME := LTIME#213503D23H33M33S709MS551US615NS;
    bLtime : LTIME := LTIME#213503D23H34M33S709MS551US615NS;

    aLword : LWORD := 16#0123456789ABCDEE;
    bLword : LWORD := 16#0123456789ABCDEF;

    aReal : REAL := 1232.5;
    bReal : REAL := 1234.4;

    aSint : SINT := -123;
    bSint : SINT := -128;

    aString : STRING := 'Hello there!';
    bString : STRING := 'Hello there';

    aTime : TIME := T#11H34M13S241MS;
    bTime : TIME := T#11H34M13S244MS;

    aTimeOfDay : TIME_OF_DAY := TIME_OF_DAY#06:21:10.492;
    bTimeOfDay : TIME_OF_DAY := TIME_OF_DAY#06:21:11.492;

    aUdint : UDINT := 21845122;
    bUdint : UDINT := 21845123;

    aUint : UINT := 65534;
    bUint : UINT := 65535;

    aUlint : ULINT := 45683838382;
    bUlint : ULINT := 45683838383;

    aUsint : USINT := 4;
    bUsint : USINT := 5;

    aWord : WORD := 16#ABCE;
    bWord : WORD := 16#ABCD;

    aSintDummy1 : SINT := 1;
    bSintDummy1 : SINT := 2;

    aSintDummy2 : SINT := 3;
    bSintDummy2 : SINT := 4;

    aSintDummy3 : SINT := 5;
    bSintDummy3 : SINT := 6;

    aSintDummy4 : SINT := 7;
    bSintDummy4 : SINT := 8;

    aSintDummy5 : SINT := 9;
    bSintDummy5 : SINT := 10;

    aSintDummy6 : SINT := 11;
    bSintDummy6 : SINT := 12;

    aSintDummy7 : SINT := 13;
    bSintDummy7 : SINT := 14;

    aSintDummy8 : SINT := 15;
    bSintDummy8 : SINT := 16;

    aSintDummy9 : SINT := 17;
    bSintDummy9 : SINT := 18;

    aSintDummy10 : SINT := 19;
    bSintDummy10 : SINT := 20;

    aSintDummy11 : SINT := 21;
    bSintDummy11 : SINT := 22;

    aSintDummy12 : SINT := 23;
    bSintDummy12 : SINT := 24;

    aSintDummy13 : SINT := 25;
    bSintDummy13 : SINT := 26;

    aSintDummy14 : SINT := 27;
    bSintDummy14 : SINT := 28;

    aSintDummy15 : SINT := 29;
    bSintDummy15 : SINT := 30;

    aSintDummy16 : SINT := 31;
    bSintDummy16 : SINT := 32;

    aSintDummy17 : SINT := 33;
    bSintDummy17 : SINT := 34;

    aSintDummy18 : SINT := 35;
    bSintDummy18 : SINT := 36;

    aSintDummy19 : SINT := 37;
    bSintDummy19 : SINT := 38;

    aSintDummy20 : SINT := 39;
    bSintDummy20 : SINT := 40;

    aSintDummy21 : SINT := 41;
    bSintDummy21 : SINT := 42;
END_VAR
TEST('TestWith44FailedAssertions');

AssertEquals(Expected := aAny,
             Actual := bAny,
             Message := 'Values differ');

AssertEquals_BOOL(Expected := aBool,
                  Actual := bBool,
                  Message := 'Values differ');

AssertEquals_BOOL(Expected := aBool2,
                  Actual := bBool2,
                  Message := 'Values differ');

AssertEquals_BYTE(Expected := aByte,
                  Actual := bByte,
                  Message := 'Values differ');

AssertEquals_DATE_AND_TIME(Expected := aDateAndTime,
                           Actual := bDateAndTime,
                           Message := 'Values differ');

AssertEquals_DATE(Expected := aDate,
                  Actual := bDate,
                  Message := 'Values differ');

AssertEquals_DINT(Expected := aDint,
                  Actual := bDint,
                  Message := 'Values differ');

AssertEquals_DWORD(Expected := aDword,
                   Actual := bDword,
                   Message := 'Values differ');

AssertEquals_INT(Expected := aInt,
                 Actual := bInt,
                 Message := 'Values differ');

AssertEquals_LINT(Expected := aLint,
                  Actual := bLint,
                  Message := 'Values differ');

AssertEquals_LREAL(Expected := aLreal,
                   Actual := bLreal,
                   Delta := 0.2,
                   Message := 'Values differ');

AssertEquals_LTIME(Expected := aLtime,
                   Actual := bLtime,
                   Message := 'Values differ');

AssertEquals_LWORD(Expected := aLword,
                   Actual := bLword,
                   Message := 'Values differ');

AssertEquals_REAL(Expected := aReal,
                  Actual := bReal,
                  Delta := 0.1,
                  Message := 'Values differ');

AssertEquals_SINT(Expected := aSint,
                  Actual := bSint,
                  Message := 'Values differ');

AssertEquals_STRING(Expected := aString,
                    Actual := bString,
                    Message := 'Values differ');

AssertEquals_TIME(Expected := aTime,
                  Actual := bTime,
                  Message := 'Values differ');

AssertEquals_TIME_OF_DAY(Expected := aTimeOfDay,
                         Actual := bTimeOfDay,
                         Message := 'Values differ');

AssertEquals_UDINT(Expected := aUdint,
                   Actual := bUdint,
                   Message := 'Values differ');

AssertEquals_UINT(Expected := aUint,
                  Actual := bUint,
                  Message := 'Values differ');

AssertEquals_ULINT(Expected := aUlint,
                   Actual := bUlint,
                   Message := 'Values differ');

AssertEquals_USINT(Expected := aUsint,
                   Actual := bUsint,
                   Message := 'Values differ');

AssertEquals_WORD(Expected := aWord,
                  Actual := bWord,
                  Message := 'Values differ');

AssertEquals_SINT(Expected := aSintDummy1,
                  Actual := bSintDummy1,
                  Message := 'Values differ');

AssertEquals_SINT(Expected := aSintDummy2,
                  Actual := bSintDummy2,
                  Message := 'Values differ');

AssertEquals_SINT(Expected := aSintDummy3,
                  Actual := bSintDummy3,
                  Message := 'Values differ');

AssertEquals_SINT(Expected := aSintDummy4,
                  Actual := bSintDummy4,
                  Message := 'Values differ');

AssertEquals_SINT(Expected := aSintDummy5,
                  Actual := bSintDummy5,
                  Message := 'Values differ');

AssertEquals_SINT(Expected := aSintDummy6,
                  Actual := bSintDummy6,
                  Message := 'Values differ');

AssertEquals_SINT(Expected := aSintDummy7,
                  Actual := bSintDummy7,
                  Message := 'Values differ');

AssertEquals_SINT(Expected := aSintDummy8,
                  Actual := bSintDummy8,
                  Message := 'Values differ');

AssertEquals_SINT(Expected := aSintDummy9,
                  Actual := bSintDummy9,
                  Message := 'Values differ');

AssertEquals_SINT(Expected := aSintDummy10,
                  Actual := bSintDummy10,
                  Message := 'Values differ');

AssertEquals_SINT(Expected := aSintDummy11,
                  Actual := bSintDummy11,
                  Message := 'Values differ');

AssertEquals_SINT(Expected := aSintDummy12,
                  Actual := bSintDummy12,
                  Message := 'Values differ');

AssertEquals_SINT(Expected := aSintDummy13,
                  Actual := bSintDummy13,
                  Message := 'Values differ');

AssertEquals_SINT(Expected := aSintDummy14,
                  Actual := bSintDummy14,
                  Message := 'Values differ');

AssertEquals_SINT(Expected := aSintDummy15,
                  Actual := bSintDummy15,
                  Message := 'Values differ');

AssertEquals_SINT(Expected := aSintDummy16,
                  Actual := bSintDummy16,
                  Message := 'Values differ');

AssertEquals_SINT(Expected := aSintDummy17,
                  Actual := bSintDummy17,
                  Message := 'Values differ');

AssertEquals_SINT(Expected := aSintDummy18,
                  Actual := bSintDummy18,
                  Message := 'Values differ');

AssertEquals_SINT(Expected := aSintDummy19,
                  Actual := bSintDummy19,
                  Message := 'Values differ');

AssertEquals_SINT(Expected := aSintDummy20,
                  Actual := bSintDummy20,
                  Message := 'Values differ');

AssertEquals_SINT(Expected := aSintDummy21,
                  Actual := bSintDummy21,
                  Message := 'Values differ');

TEST_FINISHED();
END_METHOD

METHOD PRIVATE TestWith45SuccessfulArrayAssertions
VAR
    aBool : ARRAY[1..5] OF BOOL := [TRUE, FALSE, TRUE, FALSE, TRUE];
    bBool : ARRAY[1..5] OF BOOL := [TRUE, FALSE, TRUE, FALSE, TRUE];

    aByte : ARRAY[1..3] OF BYTE := [16#FD, 16#34, 16#9E];
    bByte : ARRAY[1..3] OF BYTE := [16#FD, 16#34, 16#9E];

    aDint : ARRAY[2..7] OF DINT := [64, 98, 2147483647, -2147483648, 0, -63987538];
    bDint : ARRAY[2..7] OF DINT := [64, 98, 2147483647, -2147483648, 0, -63987538];

    aDword : ARRAY[2..3] OF DWORD := [16#6789ABCD, 16#EF012345];
    bDword : ARRAY[1..2] OF DWORD := [16#6789ABCD, 16#EF012345];

    aInt : ARRAY[-5..1] OF INT := [64, 98, -32768, 32767, 5478, -378, 42];
    bInt : ARRAY[1..7] OF INT := [64, 98, -32768, 32767, 5478, -378, 42];

    aLint : ARRAY[-1..0] OF LINT := [9_223_372_036_854_775_807, -9_223_372_036_854_775_808];
    bLint : ARRAY[4..5] OF LINT := [9_223_372_036_854_775_807, -9_223_372_036_854_775_808];

    aLreal : ARRAY[-5..1] OF LREAL := [64.0, 98.1, -32768.2, 32767.3, 5478.4, -378.5, 42.6];
    bLreal : ARRAY[1..7] OF LREAL := [64.0001, 98.0999, -32768.1995, 32767.3001, 5478.4002, -378.5003, 42.6001];

    aLreal2d : ARRAY[-5..-3,-1..0] OF LREAL := [64.0, 98.1, -32768.2, 32767.3, 5478.4, -378.5];
    bLreal2d : ARRAY[1..3,0..1] OF LREAL := [64.0001, 98.0999, -32768.1995, 32767.3001, 5478.4002, -378.5003];

    aLreal3d : ARRAY[-5..-4,-1..0,0..1] OF LREAL := [64.0, 98.1, -32768.2, 32767.3, 5478.4, -378.5, 42.6, 560344.0005];
    bLreal3d : ARRAY[1..2,4..5,6..7] OF LREAL := [64.0001, 98.0999, -32768.1995, 32767.3001, 5478.4002, -378.5003, 42.6001, 560344.0006];

    aLword : ARRAY[1..2] OF LWORD := [16#01234567890ABCDE, 16#EDCBA09876543210];
    bLword : ARRAY[1..2] OF LWORD := [16#01234567890ABCDE, 16#EDCBA09876543210];

    aReal : ARRAY[-5..1] OF REAL := [64.0, 98.1, -32768.2, 32767.3, 5478.4, -378.5, 42.6];
    bReal : ARRAY[1..7] OF REAL := [64.0001, 98.0999, -32768.1995, 32767.3001, 5478.4002, -378.5003, 42.6001];

    aReal2d : ARRAY[-5..-3,-1..0] OF REAL := [64.0, 98.1, -32768.2, 32767.3, 5478.4, -378.5];
    bReal2d : ARRAY[1..3,0..1] OF REAL := [64.0001, 98.0999, -32768.1995, 32767.3001, 5478.4002, -378.5003];

    aReal3d : ARRAY[-5..-4,-1..0,0..1] OF REAL := [64.0, 98.1, -32768.2, 32767.3, 5478.4, -378.5, 42.6, 560344.0005];
    bReal3d : ARRAY[1..2,4..5,6..7] OF REAL := [64.0001, 98.0999, -32768.1995, 32767.3001, 5478.4002, -378.5003, 42.6001, 560344.0006];

    aSint : ARRAY[0..3] OF SINT := [-128, 127, -34, 62];
    bSint : ARRAY[0..3] OF SINT := [-128, 127, -34, 62];

    aUdint : ARRAY[1..3] OF UDINT := [0, 4294967295, 5000];
    bUdint : ARRAY[1..3] OF UDINT := [0, 4294967295, 5000];

    aUint : ARRAY[0..4] OF UINT := [0, 65535, 2000, 34123, 59];
    bUint : ARRAY[0..4] OF UINT := [0, 65535, 2000, 34123, 59];

    aUlint : ARRAY[0..3] OF ULINT := [0, 18_446_744_073_709_551_615, 9_400_000_000_000, 3_213_000_444_000];
    bUlint : ARRAY[0..3] OF ULINT := [0, 18_446_744_073_709_551_615, 9_400_000_000_000, 3_213_000_444_000];

    aUsint : ARRAY[0..100] OF USINT := [42, 100(33)];
    bUsint : ARRAY[0..100] OF USINT := [42, 100(33)];

    aWord : ARRAY[1..5] OF WORD := [16#AAAA, 16#BBBB, 16#CCCC, 16#DDDD, 16#EEEE];
    bWord : ARRAY[1..5] OF WORD := [16#AAAA, 16#BBBB, 16#CCCC, 16#DDDD, 16#EEEE];

    aSintDummy1 : ARRAY[0..3] OF SINT := [-128, 127, -34, 62];
    bSintDummy1 : ARRAY[0..3] OF SINT := [-128, 127, -34, 62];

    aSintDummy2 : ARRAY[0..3] OF SINT := [-128, 127, -34, 62];
    bSintDummy2 : ARRAY[0..3] OF SINT := [-128, 127, -34, 62];

    aSintDummy3 : ARRAY[0..3] OF SINT := [-128, 127, -34, 62];
    bSintDummy3 : ARRAY[0..3] OF SINT := [-128, 127, -34, 62];

    aSintDummy4 : ARRAY[0..3] OF SINT := [-128, 127, -34, 62];
    bSintDummy4 : ARRAY[0..3] OF SINT := [-128, 127, -34, 62];

    aSintDummy5 : ARRAY[0..3] OF SINT := [-128, 127, -34, 62];
    bSintDummy5 : ARRAY[0..3] OF SINT := [-128, 127, -34, 62];

    aSintDummy6 : ARRAY[0..3] OF SINT := [-128, 127, -34, 62];
    bSintDummy6 : ARRAY[0..3] OF SINT := [-128, 127, -34, 62];

    aSintDummy7 : ARRAY[0..3] OF SINT := [-128, 127, -34, 62];
    bSintDummy7 : ARRAY[0..3] OF SINT := [-128, 127, -34, 62];

    aSintDummy8 : ARRAY[0..3] OF SINT := [-128, 127, -34, 62];
    bSintDummy8 : ARRAY[0..3] OF SINT := [-128, 127, -34, 62];

    aSintDummy9 : ARRAY[0..3] OF SINT := [-128, 127, -34, 62];
    bSintDummy9 : ARRAY[0..3] OF SINT := [-128, 127, -34, 62];

    aSintDummy10 : ARRAY[0..3] OF SINT := [-128, 127, -34, 62];
    bSintDummy10 : ARRAY[0..3] OF SINT := [-128, 127, -34, 62];

    aSintDummy11 : ARRAY[0..3] OF SINT := [-128, 127, -34, 62];
    bSintDummy11 : ARRAY[0..3] OF SINT := [-128, 127, -34, 62];

    aSintDummy12 : ARRAY[0..3] OF SINT := [-128, 127, -34, 62];
    bSintDummy12 : ARRAY[0..3] OF SINT := [-128, 127, -34, 62];

    aSintDummy13 : ARRAY[0..3] OF SINT := [-128, 127, -34, 62];
    bSintDummy13 : ARRAY[0..3] OF SINT := [-128, 127, -34, 62];

    aSintDummy14 : ARRAY[0..3] OF SINT := [-128, 127, -34, 62];
    bSintDummy14 : ARRAY[0..3] OF SINT := [-128, 127, -34, 62];

    aSintDummy15 : ARRAY[0..3] OF SINT := [-128, 127, -34, 62];
    bSintDummy15 : ARRAY[0..3] OF SINT := [-128, 127, -34, 62];

    aSintDummy16 : ARRAY[0..3] OF SINT := [-128, 127, -34, 62];
    bSintDummy16 : ARRAY[0..3] OF SINT := [-128, 127, -34, 62];

    aSintDummy17 : ARRAY[0..3] OF SINT := [-128, 127, -34, 62];
    bSintDummy17 : ARRAY[0..3] OF SINT := [-128, 127, -34, 62];

    aSintDummy18 : ARRAY[0..3] OF SINT := [-128, 127, -34, 62];
    bSintDummy18 : ARRAY[0..3] OF SINT := [-128, 127, -34, 62];

    aSintDummy19 : ARRAY[0..3] OF SINT := [-128, 127, -34, 62];
    bSintDummy19 : ARRAY[0..3] OF SINT := [-128, 127, -34, 62];

    aSintDummy20 : ARRAY[0..3] OF SINT := [-128, 127, -34, 62];
    bSintDummy20 : ARRAY[0..3] OF SINT := [-128, 127, -34, 62];

    aSintDummy21 : ARRAY[0..3] OF SINT := [-128, 127, -34, 62];
    bSintDummy21 : ARRAY[0..3] OF SINT := [-128, 127, -34, 62];

    aSintDummy22 : ARRAY[0..3] OF SINT := [-128, 127, -34, 62];
    bSintDummy22 : ARRAY[0..3] OF SINT := [-128, 127, -34, 62];

    aSintDummy23 : ARRAY[0..3] OF SINT := [-128, 127, -34, 62];
    bSintDummy23 : ARRAY[0..3] OF SINT := [-128, 127, -34, 62];

    aSintDummy24 : ARRAY[0..3] OF SINT := [-128, 127, -34, 62];
    bSintDummy24 : ARRAY[0..3] OF SINT := [-128, 127, -34, 62];

    aSintDummy25 : ARRAY[0..3] OF SINT := [-128, 127, -34, 62];
    bSintDummy25 : ARRAY[0..3] OF SINT := [-128, 127, -34, 62];

    aSintDummy26 : ARRAY[0..3] OF SINT := [-128, 127, -34, 62];
    bSintDummy26 : ARRAY[0..3] OF SINT := [-128, 127, -34, 62];
END_VAR
TEST('TestWith45SuccessfulArrayAssertions');

AssertArrayEquals_BOOL(Expecteds := aBool,
                       Actuals := bBool,
                       Message := 'Arrays differ');

AssertArrayEquals_BYTE(Expecteds := aByte,
                       Actuals := bByte,
                       Message := 'Arrays differ');

AssertArrayEquals_DINT(Expecteds := aDint,
                       Actuals := bDint,
                       Message := 'Arrays differ');

AssertArrayEquals_DWORD(Expecteds := aDword,
                        Actuals := bDword,
                        Message := 'Arrays differ');

AssertArrayEquals_INT(Expecteds := aInt,
                      Actuals := bInt,
                      Message := 'Arrays differ');

AssertArrayEquals_LINT(Expecteds := aLint,
                      Actuals := bLint,
                      Message := 'Arrays differ');

AssertArrayEquals_LREAL(Expecteds := aLreal,
                        Actuals := bLreal,
                        Delta := 0.01,
                        Message := 'Arrays differ');

AssertArray2dEquals_LREAL(Expecteds := aLreal2d,
                          Actuals := bLreal2d,
                          Delta := 0.01,
                          Message := 'Arrays differ');

AssertArray3dEquals_LREAL(Expecteds := aLreal3d,
                          Actuals := bLreal3d,
                          Delta := 0.01,
                          Message := 'Arrays differ');

AssertArrayEquals_LWORD(Expecteds := aLword,
                        Actuals := bLword,
                        Message := 'Arrays differ');

AssertArrayEquals_REAL(Expecteds := aReal,
                       Actuals := bReal,
                       Delta := 0.01,
                       Message := 'Arrays differ');

AssertArray2dEquals_REAL(Expecteds := aReal2d,
                         Actuals := bReal2d,
                         Delta := 0.01,
                         Message := 'Arrays differ');

AssertArray3dEquals_REAL(Expecteds := aReal3d,
                         Actuals := bReal3d,
                         Delta := 0.01,
                         Message := 'Arrays differ');

AssertArrayEquals_SINT(Expecteds := aSint,
                       Actuals := bSint,
                       Message := 'Arrays differ');

AssertArrayEquals_UDINT(Expecteds := aUdint,
                        Actuals := bUdint,
                        Message := 'Arrays differ');

AssertArrayEquals_UINT(Expecteds := aUint,
                       Actuals := bUint,
                       Message := 'Arrays differ');

AssertArrayEquals_ULINT(Expecteds := aUlint,
                        Actuals := bUlint,
                        Message := 'Arrays differ');

AssertArrayEquals_USINT(Expecteds := aUsint,
                        Actuals := bUsint,
                        Message := 'Arrays differ');

AssertArrayEquals_WORD(Expecteds := aWord,
                       Actuals := bWord,
                       Message := 'Arrays differ');

AssertArrayEquals_SINT(Expecteds := aSintDummy1,
                       Actuals := bSintDummy1,
                       Message := 'Arrays differ');

AssertArrayEquals_SINT(Expecteds := aSintDummy2,
                       Actuals := bSintDummy2,
                       Message := 'Arrays differ');

AssertArrayEquals_SINT(Expecteds := aSintDummy3,
                       Actuals := bSintDummy3,
                       Message := 'Arrays differ');

AssertArrayEquals_SINT(Expecteds := aSintDummy4,
                       Actuals := bSintDummy4,
                       Message := 'Arrays differ');

AssertArrayEquals_SINT(Expecteds := aSintDummy5,
                       Actuals := bSintDummy5,
                       Message := 'Arrays differ');

AssertArrayEquals_SINT(Expecteds := aSintDummy6,
                       Actuals := bSintDummy6,
                       Message := 'Arrays differ');

AssertArrayEquals_SINT(Expecteds := aSintDummy7,
                       Actuals := bSintDummy7,
                       Message := 'Arrays differ');

AssertArrayEquals_SINT(Expecteds := aSintDummy8,
                       Actuals := bSintDummy8,
                       Message := 'Arrays differ');

AssertArrayEquals_SINT(Expecteds := aSintDummy9,
                       Actuals := bSintDummy9,
                       Message := 'Arrays differ');

AssertArrayEquals_SINT(Expecteds := aSintDummy10,
                       Actuals := bSintDummy10,
                       Message := 'Arrays differ');

AssertArrayEquals_SINT(Expecteds := aSintDummy11,
                       Actuals := bSintDummy11,
                       Message := 'Arrays differ');

AssertArrayEquals_SINT(Expecteds := aSintDummy12,
                       Actuals := bSintDummy12,
                       Message := 'Arrays differ');

AssertArrayEquals_SINT(Expecteds := aSintDummy13,
                       Actuals := bSintDummy13,
                       Message := 'Arrays differ');

AssertArrayEquals_SINT(Expecteds := aSintDummy14,
                       Actuals := bSintDummy14,
                       Message := 'Arrays differ');

AssertArrayEquals_SINT(Expecteds := aSintDummy15,
                       Actuals := bSintDummy15,
                       Message := 'Arrays differ');

AssertArrayEquals_SINT(Expecteds := aSintDummy16,
                       Actuals := bSintDummy16,
                       Message := 'Arrays differ');

AssertArrayEquals_SINT(Expecteds := aSintDummy17,
                       Actuals := bSintDummy17,
                       Message := 'Arrays differ');

AssertArrayEquals_SINT(Expecteds := aSintDummy18,
                       Actuals := bSintDummy18,
                       Message := 'Arrays differ');

AssertArrayEquals_SINT(Expecteds := aSintDummy19,
                       Actuals := bSintDummy19,
                       Message := 'Arrays differ');

AssertArrayEquals_SINT(Expecteds := aSintDummy20,
                       Actuals := bSintDummy20,
                       Message := 'Arrays differ');

AssertArrayEquals_SINT(Expecteds := aSintDummy21,
                       Actuals := bSintDummy21,
                       Message := 'Arrays differ');

AssertArrayEquals_SINT(Expecteds := aSintDummy22,
                       Actuals := bSintDummy22,
                       Message := 'Arrays differ');

AssertArrayEquals_SINT(Expecteds := aSintDummy23,
                       Actuals := bSintDummy23,
                       Message := 'Arrays differ');

AssertArrayEquals_SINT(Expecteds := aSintDummy24,
                       Actuals := bSintDummy1,
                       Message := 'Arrays differ');

AssertArrayEquals_SINT(Expecteds := aSintDummy25,
                       Actuals := bSintDummy1,
                       Message := 'Arrays differ');

AssertArrayEquals_SINT(Expecteds := aSintDummy26,
                       Actuals := bSintDummy26,
                       Message := 'Arrays differ');

TEST_FINISHED();
END_METHOD

METHOD PRIVATE TestWith46FailedArrayAssertions
VAR
    aBool : ARRAY[1..4] OF BOOL := [TRUE, FALSE, TRUE, FALSE];
    bBool : ARRAY[1..5] OF BOOL := [TRUE, FALSE, TRUE, FALSE, TRUE];

    aByte : ARRAY[1..3] OF BYTE := [16#FD, 16#34, 16#9F];
    bByte : ARRAY[1..3] OF BYTE := [16#FD, 16#34, 16#9E];

    aDint : ARRAY[2..7] OF DINT := [64, 98, 2147483647, -2147483648, 0, -63987538];
    bDint : ARRAY[1..5] OF DINT := [64, 98, 2147483647, -2147483648, 0];

    aDword : ARRAY[2..3] OF DWORD := [16#6789ABCD, 16#EF012345];
    bDword : ARRAY[1..2] OF DWORD := [16#6789ABCD, 16#EF012343];

    aDword2 : ARRAY[1..2] OF DWORD := [16#6789ABCD, 16#EF012343];
    bDword2 : ARRAY[2..3] OF DWORD := [16#6789ABCD, 16#EF012345];

    aInt : ARRAY[-5..1] OF INT := [64, 95, -32768, 32767, 5478, -378, 42];
    bInt : ARRAY[1..7] OF INT := [64, 98, -32768, 32767, 5478, -378, 42];

    aLint : ARRAY[-1..-1] OF LINT := [9_223_372_036_854_775_807];
    bLint : ARRAY[4..5] OF LINT := [9_223_372_036_854_775_807, -9_223_372_036_854_775_808];

    aLreal : ARRAY[-5..1] OF LREAL := [64.0, 97.1, -32768.2, 32767.3, 5478.4, -378.5, 42.6];
    bLreal : ARRAY[1..7] OF LREAL := [64.0001, 98.0999, -32768.1995, 32767.3001, 5478.4002, -378.5003, 42.6001];

    aLreal2d : ARRAY[-5..-3,-1..0] OF LREAL := [64.0, 98.1, -32768.2, 32767.3, 5478.4, -378.5];
    bLreal2d : ARRAY[1..3,0..1] OF LREAL := [63.0001, 98.0999, -32768.1995, 32767.3001, 5478.4002, -378.5003];

    aLreal3d : ARRAY[-5..-4,-1..0,0..1] OF LREAL := [64.0, 98.1, -32768.2, 32767.3, 5478.4, -378.5, 42.6, 560344.0005];
    bLreal3d : ARRAY[1..2,4..5,6..7] OF LREAL := [64.0001, 98.0999, -32768.1995, 32767.3001, 5476.4002, -378.5003, 42.6001, 560344.0006];

    aLword : ARRAY[1..2] OF LWORD := [16#01234567890ABCDE, 16#EDCBA09876543210];
    bLword : ARRAY[1..2] OF LWORD := [16#012345678A0ABCDE, 16#EDCBA09876543210];

    aReal : ARRAY[-5..1] OF REAL := [64.0, 98.1, -32768.2, 32767.3, 5478.4, -378.5, 42.6];
    bReal : ARRAY[1..7] OF REAL := [64.0001, 98.0999, -32768.1995, 32767.3001, 5478.4002, -378.5003, 42.6001];

    aReal2d : ARRAY[-5..-3,-1..0] OF REAL := [64.0, 98.1, -32768.2, 32767.3, 5478.4, -378.5];
    bReal2d : ARRAY[1..3,0..1] OF REAL := [64.0001, 98.0999, -32761.1995, 32767.3001, 5478.4002, -378.5003];

    aReal3d : ARRAY[-5..-4,-1..0,0..1] OF REAL := [64.0, 93.1, -32768.2, 32767.3, 5478.4, -378.5, 42.6, 560344.0005];
    bReal3d : ARRAY[1..2,4..5,6..7] OF REAL := [64.0001, 98.0999, -32768.1995, 32767.3001, 5478.4002, -378.5003, 42.6001, 560344.0006];

    aSint : ARRAY[0..2] OF SINT := [-128, 127, -34];
    bSint : ARRAY[0..3] OF SINT := [-128, 127, -34, 62];

    aUdint : ARRAY[1..3] OF UDINT := [0, 4294967295, 5000];
    bUdint : ARRAY[1..1] OF UDINT := [0];

    aUint : ARRAY[0..4] OF UINT := [0, 65535, 2001, 34123, 59];
    bUint : ARRAY[0..4] OF UINT := [0, 65535, 2000, 34123, 59];

    aUlint : ARRAY[0..3] OF ULINT := [0, 18_446_744_073_709_551_614, 9_400_000_000_000, 3_213_000_444_000];
    bUlint : ARRAY[0..3] OF ULINT := [0, 18_446_744_073_709_551_615, 9_400_000_000_000, 3_213_000_444_000];

    aUsint : ARRAY[0..99] OF USINT := [42, 99(33)];
    bUsint : ARRAY[0..100] OF USINT := [42, 100(33)];

    aWord : ARRAY[1..5] OF WORD := [16#AAAA, 16#BBBF, 16#CCCC, 16#DDDD, 16#EEEE];
    bWord : ARRAY[1..5] OF WORD := [16#AAAA, 16#BBBB, 16#CCCC, 16#DDDD, 16#EEEE];
    

    aSintDummy1 : ARRAY[0..3] OF SINT := [-128, 127, -34, 62];
    bSintDummy1 : ARRAY[0..3] OF SINT := [-128, 127, -34, 63];

    aSintDummy2 : ARRAY[0..3] OF SINT := [-128, 127, -34, 64];
    bSintDummy2 : ARRAY[0..3] OF SINT := [-128, 127, -34, 65];

    aSintDummy3 : ARRAY[0..3] OF SINT := [-128, 127, -34, 66];
    bSintDummy3 : ARRAY[0..3] OF SINT := [-128, 127, -34, 67];

    aSintDummy4 : ARRAY[0..3] OF SINT := [-128, 127, -34, 68];
    bSintDummy4 : ARRAY[0..3] OF SINT := [-128, 127, -34, 69];

    aSintDummy5 : ARRAY[0..3] OF SINT := [-128, 127, -34, 70];
    bSintDummy5 : ARRAY[0..3] OF SINT := [-128, 127, -34, 71];

    aSintDummy6 : ARRAY[0..3] OF SINT := [-128, 127, -34, 72];
    bSintDummy6 : ARRAY[0..3] OF SINT := [-128, 127, -34, 73];

    aSintDummy7 : ARRAY[0..3] OF SINT := [-128, 127, -34, 74];
    bSintDummy7 : ARRAY[0..3] OF SINT := [-128, 127, -34, 75];

    aSintDummy8 : ARRAY[0..3] OF SINT := [-128, 127, -34, 76];
    bSintDummy8 : ARRAY[0..3] OF SINT := [-128, 127, -34, 77];

    aSintDummy9 : ARRAY[0..3] OF SINT := [-128, 127, -34, 78];
    bSintDummy9 : ARRAY[0..3] OF SINT := [-128, 127, -34, 79];

    aSintDummy10 : ARRAY[0..3] OF SINT := [-128, 127, -34, 80];
    bSintDummy10 : ARRAY[0..3] OF SINT := [-128, 127, -34, 81];

    aSintDummy11 : ARRAY[0..3] OF SINT := [-128, 127, -34, 82];
    bSintDummy11 : ARRAY[0..3] OF SINT := [-128, 127, -34, 83];

    aSintDummy12 : ARRAY[0..3] OF SINT := [-128, 127, -34, 84];
    bSintDummy12 : ARRAY[0..3] OF SINT := [-128, 127, -34, 85];

    aSintDummy13 : ARRAY[0..3] OF SINT := [-128, 127, -34, 86];
    bSintDummy13 : ARRAY[0..3] OF SINT := [-128, 127, -34, 87];

    aSintDummy14 : ARRAY[0..3] OF SINT := [-128, 127, -34, 88];
    bSintDummy14 : ARRAY[0..3] OF SINT := [-128, 127, -34, 89];

    aSintDummy15 : ARRAY[0..3] OF SINT := [-128, 127, -34, 90];
    bSintDummy15 : ARRAY[0..3] OF SINT := [-128, 127, -34, 91];

    aSintDummy16 : ARRAY[0..3] OF SINT := [-128, 127, -34, 92];
    bSintDummy16 : ARRAY[0..3] OF SINT := [-128, 127, -34, 93];

    aSintDummy17 : ARRAY[0..3] OF SINT := [-128, 127, -34, 94];
    bSintDummy17 : ARRAY[0..3] OF SINT := [-128, 127, -34, 95];

    aSintDummy18 : ARRAY[0..3] OF SINT := [-128, 127, -34, 96];
    bSintDummy18 : ARRAY[0..3] OF SINT := [-128, 127, -34, 97];

    aSintDummy19 : ARRAY[0..3] OF SINT := [-128, 127, -34, 98];
    bSintDummy19 : ARRAY[0..3] OF SINT := [-128, 127, -34, 99];

    aSintDummy20 : ARRAY[0..3] OF SINT := [-128, 127, -34, 100];
    bSintDummy20 : ARRAY[0..3] OF SINT := [-128, 127, -34, 101];

    aSintDummy21 : ARRAY[0..3] OF SINT := [-128, 127, -34, 102];
    bSintDummy21 : ARRAY[0..3] OF SINT := [-128, 127, -34, 103];

